LIN {X 87.779,Y 86.082,Z 65.500,A 180.000,B 0.000,C 180.000} C_DIS
LIN {X 87.601,Y 86.233,Z 65.500,A 180.000,B 0.000,C 180.000} C_DIS
LIN {X 87.468,Y 86.349,Z 65.500,A 180.000,B 0.000,C 180.000} C_DIS
LIN {X 87.422,Y 86.393,Z 65.500,A 180.000,B 0.000,C 180.000} C_DIS
LIN {X 87.064,Y 86.731,Z 65.500,A 180.000,B 0.000,C 180.000} C_DIS
LIN {X 86.901,Y 86.885,Z 65.500,A 180.000,B 0.000,C 180.000} C_DIS
LIN {X 86.885,Y 86.901,Z 65.500,A 180.000,B 0.000,C 180.000} C_DIS
LIN {X 86.731,Y 87.064,Z 65.500,A 180.000,B 0.000,C 180.000} C_DIS
LIN {X 86.393,Y 87.422,Z 65.500,A 180.000,B 0.000,C 180.000} C_DIS
LIN {X 86.349,Y 87.468,Z 65.500,A 180.000,B 0.000,C 180.000} C_DIS
LIN {X 86.233,Y 87.601,Z 65.500,A 180.000,B 0.000,C 180.000} C_DIS
LIN {X 85.931,Y 87.958,Z 65.500,A 180.000,B 0.000,C 180.000} C_DIS
LIN {X 85.813,Y 88.098,Z 65.500,A 180.000,B 0.000,C 180.000} C_DIS
LIN {X 85.781,Y 88.137,Z 65.500,A 180.000,B 0.000,C 180.000} C_DIS
LIN {X 85.645,Y 88.316,Z 65.500,A 180.000,B 0.000,C 180.000} C_DIS
LIN {X 85.376,Y 88.673,Z 65.500,A 180.000,B 0.000,C 180.000} C_DIS
LIN {X 85.276,Y 88.806,Z 65.500,A 180.000,B 0.000,C 180.000} C_DIS
LIN {X 85.244,Y 88.852,Z 65.500,A 180.000,B 0.000,C 180.000} C_DIS
LIN {X 85.125,Y 89.031,Z 65.500,A 180.000,B 0.000,C 180.000} C_DIS
LIN {X 84.886,Y 89.388,Z 65.500,A 180.000,B 0.000,C 180.000} C_DIS
LIN {X 84.770,Y 89.567,Z 65.500,A 180.000,B 0.000,C 180.000} C_DIS
LIN {X 84.740,Y 89.618,Z 65.500,A 180.000,B 0.000,C 180.000} C_DIS
LIN {X 84.454,Y 90.103,Z 65.500,A 180.000,B 0.000,C 180.000} C_DIS
LIN {X 84.383,Y 90.225,Z 65.500,A 180.000,B 0.000,C 180.000} C_DIS
LIN {X 84.351,Y 90.282,Z 65.500,A 180.000,B 0.000,C 180.000} C_DIS
LIN {X 84.259,Y 90.461,Z 65.500,A 180.000,B 0.000,C 180.000} C_DIS
LIN {X 84.025,Y 90.913,Z 65.500,A 180.000,B 0.000,C 180.000} C_DIS
LIN {X 83.983,Y 90.997,Z 65.500,A 180.000,B 0.000,C 180.000} C_DIS
LIN {X 83.902,Y 91.176,Z 65.500,A 180.000,B 0.000,C 180.000} C_DIS
LIN {X 83.668,Y 91.700,Z 65.500,A 180.000,B 0.000,C 180.000} C_DIS
LIN {X 83.662,Y 91.712,Z 65.500,A 180.000,B 0.000,C 180.000} C_DIS
LIN {X 83.591,Y 91.891,Z 65.500,A 180.000,B 0.000,C 180.000} C_DIS
LIN {X 83.386,Y 92.427,Z 65.500,A 180.000,B 0.000,C 180.000} C_DIS
LIN {X 83.322,Y 92.606,Z 65.500,A 180.000,B 0.000,C 180.000} C_DIS
LIN {X 83.310,Y 92.642,Z 65.500,A 180.000,B 0.000,C 180.000} C_DIS
LIN {X 83.131,Y 93.203,Z 65.500,A 180.000,B 0.000,C 180.000} C_DIS
LIN {X 83.094,Y 93.321,Z 65.500,A 180.000,B 0.000,C 180.000} C_DIS
LIN {X 83.046,Y 93.500,Z 65.500,A 180.000,B 0.000,C 180.000} C_DIS
LIN {X 82.908,Y 94.036,Z 65.500,A 180.000,B 0.000,C 180.000} C_DIS
LIN {X 82.865,Y 94.215,Z 65.500,A 180.000,B 0.000,C 180.000} C_DIS
LIN {X 82.829,Y 94.394,Z 65.500,A 180.000,B 0.000,C 180.000} C_DIS
LIN {X 82.758,Y 94.751,Z 65.500,A 180.000,B 0.000,C 180.000} C_DIS
LIN {X 82.722,Y 94.930,Z 65.500,A 180.000,B 0.000,C 180.000} C_DIS
LIN {X 82.694,Y 95.109,Z 65.500,A 180.000,B 0.000,C 180.000} C_DIS
LIN {X 82.618,Y 95.645,Z 65.500,A 180.000,B 0.000,C 180.000} C_DIS
LIN {X 82.595,Y 95.815,Z 65.500,A 180.000,B 0.000,C 180.000} C_DIS
LIN {X 82.594,Y 95.824,Z 65.500,A 180.000,B 0.000,C 180.000} C_DIS
LIN {X 82.578,Y 96.003,Z 65.500,A 180.000,B 0.000,C 180.000} C_DIS
LIN {X 82.533,Y 96.539,Z 65.500,A 180.000,B 0.000,C 180.000} C_DIS
LIN {X 82.521,Y 96.718,Z 65.500,A 180.000,B 0.000,C 180.000} C_DIS
LIN {X 82.516,Y 96.897,Z 65.500,A 180.000,B 0.000,C 180.000} C_DIS
LIN {X 82.501,Y 97.433,Z 65.500,A 180.000,B 0.000,C 180.000} C_DIS
LIN {X 82.502,Y 97.612,Z 65.500,A 180.000,B 0.000,C 180.000} C_DIS
LIN {X 82.517,Y 98.148,Z 65.500,A 180.000,B 0.000,C 180.000} C_DIS
LIN {X 82.523,Y 98.327,Z 65.500,A 180.000,B 0.000,C 180.000} C_DIS
LIN {X 82.536,Y 98.505,Z 65.500,A 180.000,B 0.000,C 180.000} C_DIS
LIN {X 82.582,Y 99.042,Z 65.500,A 180.000,B 0.000,C 180.000} C_DIS
LIN {X 82.595,Y 99.185,Z 65.500,A 180.000,B 0.000,C 180.000} C_DIS
LIN {X 82.599,Y 99.221,Z 65.500,A 180.000,B 0.000,C 180.000} C_DIS
LIN {X 82.624,Y 99.399,Z 65.500,A 180.000,B 0.000,C 180.000} C_DIS
LIN {X 82.700,Y 99.936,Z 65.500,A 180.000,B 0.000,C 180.000} C_DIS
LIN {X 82.731,Y 100.114,Z 65.500,A 180.000,B 0.000,C 180.000} C_DIS
LIN {X 82.838,Y 100.651,Z 65.500,A 180.000,B 0.000,C 180.000} C_DIS
LIN {X 82.874,Y 100.829,Z 65.500,A 180.000,B 0.000,C 180.000} C_DIS
LIN {X 82.919,Y 101.008,Z 65.500,A 180.000,B 0.000,C 180.000} C_DIS
LIN {X 83.057,Y 101.545,Z 65.500,A 180.000,B 0.000,C 180.000} C_DIS
LIN {X 83.108,Y 101.723,Z 65.500,A 180.000,B 0.000,C 180.000} C_DIS
LIN {X 83.310,Y 102.358,Z 65.500,A 180.000,B 0.000,C 180.000} C_DIS
LIN {X 83.336,Y 102.438,Z 65.500,A 180.000,B 0.000,C 180.000} C_DIS
LIN {X 83.403,Y 102.617,Z 65.500,A 180.000,B 0.000,C 180.000} C_DIS
LIN {X 83.608,Y 103.153,Z 65.500,A 180.000,B 0.000,C 180.000} C_DIS
LIN {X 83.668,Y 103.300,Z 65.500,A 180.000,B 0.000,C 180.000} C_DIS
LIN {X 83.922,Y 103.869,Z 65.500,A 180.000,B 0.000,C 180.000} C_DIS
LIN {X 84.005,Y 104.047,Z 65.500,A 180.000,B 0.000,C 180.000} C_DIS
LIN {X 84.025,Y 104.087,Z 65.500,A 180.000,B 0.000,C 180.000} C_DIS
LIN {X 84.282,Y 104.584,Z 65.500,A 180.000,B 0.000,C 180.000} C_DIS
LIN {X 84.375,Y 104.762,Z 65.500,A 180.000,B 0.000,C 180.000} C_DIS
LIN {X 84.383,Y 104.775,Z 65.500,A 180.000,B 0.000,C 180.000} C_DIS
LIN {X 84.480,Y 104.941,Z 65.500,A 180.000,B 0.000,C 180.000} C_DIS
LIN {X 84.740,Y 105.382,Z 65.500,A 180.000,B 0.000,C 180.000} C_DIS
LIN {X 84.797,Y 105.477,Z 65.500,A 180.000,B 0.000,C 180.000} C_DIS
LIN {X 84.915,Y 105.656,Z 65.500,A 180.000,B 0.000,C 180.000} C_DIS
LIN {X 85.154,Y 106.014,Z 65.500,A 180.000,B 0.000,C 180.000} C_DIS
LIN {X 85.276,Y 106.193,Z 65.500,A 180.000,B 0.000,C 180.000} C_DIS
LIN {X 85.276,Y 106.194,Z 65.500,A 180.000,B 0.000,C 180.000} C_DIS
LIN {X 85.409,Y 106.371,Z 65.500,A 180.000,B 0.000,C 180.000} C_DIS
LIN {X 85.678,Y 106.729,Z 65.500,A 180.000,B 0.000,C 180.000} C_DIS
LIN {X 85.813,Y 106.902,Z 65.500,A 180.000,B 0.000,C 180.000} C_DIS
LIN {X 85.818,Y 106.908,Z 65.500,A 180.000,B 0.000,C 180.000} C_DIS
LIN {X 86.271,Y 107.444,Z 65.500,A 180.000,B 0.000,C 180.000} C_DIS
LIN {X 86.349,Y 107.532,Z 65.500,A 180.000,B 0.000,C 180.000} C_DIS
LIN {X 86.435,Y 107.623,Z 65.500,A 180.000,B 0.000,C 180.000} C_DIS
LIN {X 86.773,Y 107.980,Z 65.500,A 180.000,B 0.000,C 180.000} C_DIS
LIN {X 86.885,Y 108.099,Z 65.500,A 180.000,B 0.000,C 180.000} C_DIS
LIN {X 86.947,Y 108.159,Z 65.500,A 180.000,B 0.000,C 180.000} C_DIS
LIN {X 87.422,Y 108.607,Z 65.500,A 180.000,B 0.000,C 180.000} C_DIS
LIN {X 87.517,Y 108.695,Z 65.500,A 180.000,B 0.000,C 180.000} C_DIS
LIN {X 87.601,Y 108.767,Z 65.500,A 180.000,B 0.000,C 180.000} C_DIS
LIN {X 87.958,Y 109.069,Z 65.500,A 180.000,B 0.000,C 180.000} C_DIS
LIN {X 88.137,Y 109.219,Z 65.500,A 180.000,B 0.000,C 180.000} C_DIS
LIN {X 88.153,Y 109.232,Z 65.500,A 180.000,B 0.000,C 180.000} C_DIS
LIN {X 88.316,Y 109.355,Z 65.500,A 180.000,B 0.000,C 180.000} C_DIS
LIN {X 88.673,Y 109.624,Z 65.500,A 180.000,B 0.000,C 180.000} C_DIS
LIN {X 88.852,Y 109.756,Z 65.500,A 180.000,B 0.000,C 180.000} C_DIS
LIN {X 88.870,Y 109.768,Z 65.500,A 180.000,B 0.000,C 180.000} C_DIS
LIN {X 89.031,Y 109.875,Z 65.500,A 180.000,B 0.000,C 180.000} C_DIS
LIN {X 89.405,Y 110.126,Z 65.500,A 180.000,B 0.000,C 180.000} C_DIS
LIN {X 89.567,Y 110.230,Z 65.500,A 180.000,B 0.000,C 180.000} C_DIS
LIN {X 89.693,Y 110.304,Z 65.500,A 180.000,B 0.000,C 180.000} C_DIS
LIN {X 90.103,Y 110.546,Z 65.500,A 180.000,B 0.000,C 180.000} C_DIS
LIN {X 90.282,Y 110.649,Z 65.500,A 180.000,B 0.000,C 180.000} C_DIS
LIN {X 90.307,Y 110.662,Z 65.500,A 180.000,B 0.000,C 180.000} C_DIS
LIN {X 90.818,Y 110.926,Z 65.500,A 180.000,B 0.000,C 180.000} C_DIS
LIN {X 90.997,Y 111.017,Z 65.500,A 180.000,B 0.000,C 180.000} C_DIS
LIN {X 91.002,Y 111.019,Z 65.500,A 180.000,B 0.000,C 180.000} C_DIS
LIN {X 91.176,Y 111.098,Z 65.500,A 180.000,B 0.000,C 180.000} C_DIS
LIN {X 91.533,Y 111.258,Z 65.500,A 180.000,B 0.000,C 180.000} C_DIS
LIN {X 91.712,Y 111.338,Z 65.500,A 180.000,B 0.000,C 180.000} C_DIS
LIN {X 91.806,Y 111.377,Z 65.500,A 180.000,B 0.000,C 180.000} C_DIS
LIN {X 91.891,Y 111.409,Z 65.500,A 180.000,B 0.000,C 180.000} C_DIS
LIN {X 92.427,Y 111.614,Z 65.500,A 180.000,B 0.000,C 180.000} C_DIS
LIN {X 92.606,Y 111.678,Z 65.500,A 180.000,B 0.000,C 180.000} C_DIS
LIN {X 92.964,Y 111.792,Z 65.500,A 180.000,B 0.000,C 180.000} C_DIS
LIN {X 93.142,Y 111.849,Z 65.500,A 180.000,B 0.000,C 180.000} C_DIS
LIN {X 93.321,Y 111.906,Z 65.500,A 180.000,B 0.000,C 180.000} C_DIS
LIN {X 93.346,Y 111.913,Z 65.500,A 180.000,B 0.000,C 180.000} C_DIS
LIN {X 93.500,Y 111.954,Z 65.500,A 180.000,B 0.000,C 180.000} C_DIS
LIN {X 94.036,Y 112.092,Z 65.500,A 180.000,B 0.000,C 180.000} C_DIS
LIN {X 94.215,Y 112.135,Z 65.500,A 180.000,B 0.000,C 180.000} C_DIS
LIN {X 94.394,Y 112.171,Z 65.500,A 180.000,B 0.000,C 180.000} C_DIS
LIN {X 94.895,Y 112.271,Z 65.500,A 180.000,B 0.000,C 180.000} C_DIS
LIN {X 94.930,Y 112.278,Z 65.500,A 180.000,B 0.000,C 180.000} C_DIS
LIN {X 95.109,Y 112.306,Z 65.500,A 180.000,B 0.000,C 180.000} C_DIS
LIN {X 95.645,Y 112.382,Z 65.500,A 180.000,B 0.000,C 180.000} C_DIS
LIN {X 95.824,Y 112.406,Z 65.500,A 180.000,B 0.000,C 180.000} C_DIS
LIN {X 96.003,Y 112.422,Z 65.500,A 180.000,B 0.000,C 180.000} C_DIS
LIN {X 96.539,Y 112.467,Z 65.500,A 180.000,B 0.000,C 180.000} C_DIS
LIN {X 96.718,Y 112.479,Z 65.500,A 180.000,B 0.000,C 180.000} C_DIS
LIN {X 96.897,Y 112.484,Z 65.500,A 180.000,B 0.000,C 180.000} C_DIS
LIN {X 97.433,Y 112.499,Z 65.500,A 180.000,B 0.000,C 180.000} C_DIS
LIN {X 97.612,Y 112.498,Z 65.500,A 180.000,B 0.000,C 180.000} C_DIS
LIN {X 98.148,Y 112.483,Z 65.500,A 180.000,B 0.000,C 180.000} C_DIS
LIN {X 98.327,Y 112.477,Z 65.500,A 180.000,B 0.000,C 180.000} C_DIS
LIN {X 98.505,Y 112.464,Z 65.500,A 180.000,B 0.000,C 180.000} C_DIS
LIN {X 99.042,Y 112.418,Z 65.500,A 180.000,B 0.000,C 180.000} C_DIS
LIN {X 99.221,Y 112.401,Z 65.500,A 180.000,B 0.000,C 180.000} C_DIS
LIN {X 99.399,Y 112.376,Z 65.500,A 180.000,B 0.000,C 180.000} C_DIS
LIN {X 99.936,Y 112.300,Z 65.500,A 180.000,B 0.000,C 180.000} C_DIS
LIN {X 100.105,Y 112.271,Z 65.500,A 180.000,B 0.000,C 180.000} C_DIS
LIN {X 100.651,Y 112.162,Z 65.500,A 180.000,B 0.000,C 180.000} C_DIS
LIN {X 100.829,Y 112.126,Z 65.500,A 180.000,B 0.000,C 180.000} C_DIS
LIN {X 100.966,Y 112.092,Z 65.500,A 180.000,B 0.000,C 180.000} C_DIS
LIN {X 101.545,Y 111.943,Z 65.500,A 180.000,B 0.000,C 180.000} C_DIS
LIN {X 101.654,Y 111.913,Z 65.500,A 180.000,B 0.000,C 180.000} C_DIS
LIN {X 101.723,Y 111.892,Z 65.500,A 180.000,B 0.000,C 180.000} C_DIS
LIN {X 102.260,Y 111.721,Z 65.500,A 180.000,B 0.000,C 180.000} C_DIS
LIN {X 102.438,Y 111.664,Z 65.500,A 180.000,B 0.000,C 180.000} C_DIS
LIN {X 102.617,Y 111.597,Z 65.500,A 180.000,B 0.000,C 180.000} C_DIS
LIN {X 103.153,Y 111.392,Z 65.500,A 180.000,B 0.000,C 180.000} C_DIS
LIN {X 103.194,Y 111.377,Z 65.500,A 180.000,B 0.000,C 180.000} C_DIS
LIN {X 103.332,Y 111.318,Z 65.500,A 180.000,B 0.000,C 180.000} C_DIS
LIN {X 103.869,Y 111.078,Z 65.500,A 180.000,B 0.000,C 180.000} C_DIS
LIN {X 103.998,Y 111.019,Z 65.500,A 180.000,B 0.000,C 180.000} C_DIS
LIN {X 104.047,Y 110.995,Z 65.500,A 180.000,B 0.000,C 180.000} C_DIS
LIN {X 104.226,Y 110.903,Z 65.500,A 180.000,B 0.000,C 180.000} C_DIS
LIN {X 104.693,Y 110.662,Z 65.500,A 180.000,B 0.000,C 180.000} C_DIS
LIN {X 104.762,Y 110.625,Z 65.500,A 180.000,B 0.000,C 180.000} C_DIS
LIN {X 104.941,Y 110.520,Z 65.500,A 180.000,B 0.000,C 180.000} C_DIS
LIN {X 105.307,Y 110.304,Z 65.500,A 180.000,B 0.000,C 180.000} C_DIS
LIN {X 105.477,Y 110.203,Z 65.500,A 180.000,B 0.000,C 180.000} C_DIS
LIN {X 105.595,Y 110.126,Z 65.500,A 180.000,B 0.000,C 180.000} C_DIS
LIN {X 106.014,Y 109.846,Z 65.500,A 180.000,B 0.000,C 180.000} C_DIS
LIN {X 106.130,Y 109.768,Z 65.500,A 180.000,B 0.000,C 180.000} C_DIS
LIN {X 106.193,Y 109.724,Z 65.500,A 180.000,B 0.000,C 180.000} C_DIS
LIN {X 106.371,Y 109.591,Z 65.500,A 180.000,B 0.000,C 180.000} C_DIS
LIN {X 106.729,Y 109.322,Z 65.500,A 180.000,B 0.000,C 180.000} C_DIS
LIN {X 106.847,Y 109.232,Z 65.500,A 180.000,B 0.000,C 180.000} C_DIS
LIN {X 106.908,Y 109.182,Z 65.500,A 180.000,B 0.000,C 180.000} C_DIS
LIN {X 107.444,Y 108.729,Z 65.500,A 180.000,B 0.000,C 180.000} C_DIS
LIN {X 107.483,Y 108.695,Z 65.500,A 180.000,B 0.000,C 180.000} C_DIS
LIN {X 107.623,Y 108.565,Z 65.500,A 180.000,B 0.000,C 180.000} C_DIS
LIN {X 108.053,Y 108.159,Z 65.500,A 180.000,B 0.000,C 180.000} C_DIS
LIN {X 108.159,Y 108.053,Z 65.500,A 180.000,B 0.000,C 180.000} C_DIS
LIN {X 108.565,Y 107.623,Z 65.500,A 180.000,B 0.000,C 180.000} C_DIS
LIN {X 108.695,Y 107.483,Z 65.500,A 180.000,B 0.000,C 180.000} C_DIS
LIN {X 108.729,Y 107.444,Z 65.500,A 180.000,B 0.000,C 180.000} C_DIS
LIN {X 109.182,Y 106.908,Z 65.500,A 180.000,B 0.000,C 180.000} C_DIS
LIN {X 109.232,Y 106.847,Z 65.500,A 180.000,B 0.000,C 180.000} C_DIS
LIN {X 109.322,Y 106.729,Z 65.500,A 180.000,B 0.000,C 180.000} C_DIS
LIN {X 109.591,Y 106.371,Z 65.500,A 180.000,B 0.000,C 180.000} C_DIS
LIN {X 109.724,Y 106.193,Z 65.500,A 180.000,B 0.000,C 180.000} C_DIS
LIN {X 109.768,Y 106.130,Z 65.500,A 180.000,B 0.000,C 180.000} C_DIS
LIN {X 109.846,Y 106.014,Z 65.500,A 180.000,B 0.000,C 180.000} C_DIS
LIN {X 110.126,Y 105.595,Z 65.500,A 180.000,B 0.000,C 180.000} C_DIS
LIN {X 110.203,Y 105.477,Z 65.500,A 180.000,B 0.000,C 180.000} C_DIS
LIN {X 110.304,Y 105.307,Z 65.500,A 180.000,B 0.000,C 180.000} C_DIS
LIN {X 110.520,Y 104.941,Z 65.500,A 180.000,B 0.000,C 180.000} C_DIS
LIN {X 110.625,Y 104.762,Z 65.500,A 180.000,B 0.000,C 180.000} C_DIS
LIN {X 110.662,Y 104.693,Z 65.500,A 180.000,B 0.000,C 180.000} C_DIS
LIN {X 110.903,Y 104.226,Z 65.500,A 180.000,B 0.000,C 180.000} C_DIS
LIN {X 110.995,Y 104.047,Z 65.500,A 180.000,B 0.000,C 180.000} C_DIS
LIN {X 111.019,Y 103.998,Z 65.500,A 180.000,B 0.000,C 180.000} C_DIS
LIN {X 111.078,Y 103.869,Z 65.500,A 180.000,B 0.000,C 180.000} C_DIS
LIN {X 111.318,Y 103.332,Z 65.500,A 180.000,B 0.000,C 180.000} C_DIS
LIN {X 111.377,Y 103.194,Z 65.500,A 180.000,B 0.000,C 180.000} C_DIS
LIN {X 111.392,Y 103.153,Z 65.500,A 180.000,B 0.000,C 180.000} C_DIS
LIN {X 111.597,Y 102.617,Z 65.500,A 180.000,B 0.000,C 180.000} C_DIS
LIN {X 111.664,Y 102.438,Z 65.500,A 180.000,B 0.000,C 180.000} C_DIS
LIN {X 111.721,Y 102.260,Z 65.500,A 180.000,B 0.000,C 180.000} C_DIS
LIN {X 111.892,Y 101.723,Z 65.500,A 180.000,B 0.000,C 180.000} C_DIS
LIN {X 111.913,Y 101.654,Z 65.500,A 180.000,B 0.000,C 180.000} C_DIS
LIN {X 111.943,Y 101.545,Z 65.500,A 180.000,B 0.000,C 180.000} C_DIS
LIN {X 112.092,Y 100.966,Z 65.500,A 180.000,B 0.000,C 180.000} C_DIS
LIN {X 112.126,Y 100.829,Z 65.500,A 180.000,B 0.000,C 180.000} C_DIS
LIN {X 112.162,Y 100.651,Z 65.500,A 180.000,B 0.000,C 180.000} C_DIS
LIN {X 112.271,Y 100.105,Z 65.500,A 180.000,B 0.000,C 180.000} C_DIS
LIN {X 112.300,Y 99.936,Z 65.500,A 180.000,B 0.000,C 180.000} C_DIS
LIN {X 112.376,Y 99.399,Z 65.500,A 180.000,B 0.000,C 180.000} C_DIS
LIN {X 112.401,Y 99.221,Z 65.500,A 180.000,B 0.000,C 180.000} C_DIS
LIN {X 112.418,Y 99.042,Z 65.500,A 180.000,B 0.000,C 180.000} C_DIS
LIN {X 112.464,Y 98.505,Z 65.500,A 180.000,B 0.000,C 180.000} C_DIS
LIN {X 112.477,Y 98.327,Z 65.500,A 180.000,B 0.000,C 180.000} C_DIS
LIN {X 112.483,Y 98.148,Z 65.500,A 180.000,B 0.000,C 180.000} C_DIS
LIN {X 112.498,Y 97.612,Z 65.500,A 180.000,B 0.000,C 180.000} C_DIS
LIN {X 112.499,Y 97.433,Z 65.500,A 180.000,B 0.000,C 180.000} C_DIS
LIN {X 112.484,Y 96.897,Z 65.500,A 180.000,B 0.000,C 180.000} C_DIS
LIN {X 112.479,Y 96.718,Z 65.500,A 180.000,B 0.000,C 180.000} C_DIS
LIN {X 112.467,Y 96.539,Z 65.500,A 180.000,B 0.000,C 180.000} C_DIS
LIN {X 112.422,Y 96.003,Z 65.500,A 180.000,B 0.000,C 180.000} C_DIS
LIN {X 112.406,Y 95.824,Z 65.500,A 180.000,B 0.000,C 180.000} C_DIS
LIN {X 112.382,Y 95.645,Z 65.500,A 180.000,B 0.000,C 180.000} C_DIS
LIN {X 112.306,Y 95.109,Z 65.500,A 180.000,B 0.000,C 180.000} C_DIS
LIN {X 112.278,Y 94.930,Z 65.500,A 180.000,B 0.000,C 180.000} C_DIS
LIN {X 112.271,Y 94.895,Z 65.500,A 180.000,B 0.000,C 180.000} C_DIS
LIN {X 112.171,Y 94.394,Z 65.500,A 180.000,B 0.000,C 180.000} C_DIS
LIN {X 112.135,Y 94.215,Z 65.500,A 180.000,B 0.000,C 180.000} C_DIS
LIN {X 112.092,Y 94.036,Z 65.500,A 180.000,B 0.000,C 180.000} C_DIS
LIN {X 111.954,Y 93.500,Z 65.500,A 180.000,B 0.000,C 180.000} C_DIS
LIN {X 111.913,Y 93.346,Z 65.500,A 180.000,B 0.000,C 180.000} C_DIS
LIN {X 111.906,Y 93.321,Z 65.500,A 180.000,B 0.000,C 180.000} C_DIS
LIN {X 111.849,Y 93.142,Z 65.500,A 180.000,B 0.000,C 180.000} C_DIS
LIN {X 111.734,Y 92.782,Z 65.500,A 180.000,B 0.000,C 180.000} C_DIS
LIN {X 111.678,Y 92.606,Z 65.500,A 180.000,B 0.000,C 180.000} C_DIS
LIN {X 111.614,Y 92.427,Z 65.500,A 180.000,B 0.000,C 180.000} C_DIS
LIN {X 111.409,Y 91.891,Z 65.500,A 180.000,B 0.000,C 180.000} C_DIS
LIN {X 111.377,Y 91.806,Z 65.500,A 180.000,B 0.000,C 180.000} C_DIS
LIN {X 111.338,Y 91.712,Z 65.500,A 180.000,B 0.000,C 180.000} C_DIS
LIN {X 111.258,Y 91.533,Z 65.500,A 180.000,B 0.000,C 180.000} C_DIS
LIN {X 111.098,Y 91.176,Z 65.500,A 180.000,B 0.000,C 180.000} C_DIS
LIN {X 111.019,Y 91.002,Z 65.500,A 180.000,B 0.000,C 180.000} C_DIS
LIN {X 111.017,Y 90.997,Z 65.500,A 180.000,B 0.000,C 180.000} C_DIS
LIN {X 110.946,Y 90.857,Z 65.500,A 180.000,B 0.000,C 180.000} C_DIS
; Link Move Starts
LIN {X 110.802,Y 90.577,Z 65.500,A 180.000,B 0.000,C 180.000} C_DIS
LIN {X 110.657,Y 90.297,Z 65.499,A 180.000,B 0.000,C 180.000} C_DIS
LIN {X 110.500,Y 90.024,Z 65.498,A 180.000,B 0.000,C 180.000} C_DIS
LIN {X 110.340,Y 89.753,Z 65.496,A 180.000,B 0.000,C 180.000} C_DIS
LIN {X 110.178,Y 89.483,Z 65.494,A 180.000,B 0.000,C 180.000} C_DIS
LIN {X 110.003,Y 89.221,Z 65.491,A 180.000,B 0.000,C 180.000} C_DIS
LIN {X 109.828,Y 88.959,Z 65.488,A 180.000,B 0.000,C 180.000} C_DIS
LIN {X 109.646,Y 88.702,Z 65.485,A 180.000,B 0.000,C 180.000} C_DIS
LIN {X 109.457,Y 88.450,Z 65.481,A 180.000,B 0.000,C 180.000} C_DIS
LIN {X 109.267,Y 88.199,Z 65.477,A 180.000,B 0.000,C 180.000} C_DIS
LIN {X 109.067,Y 87.956,Z 65.472,A 180.000,B 0.000,C 180.000} C_DIS
LIN {X 108.965,Y 87.835,Z 65.469,A 180.000,B 0.000,C 180.000} C_DIS
LIN {X 108.863,Y 87.715,Z 65.467,A 180.000,B 0.000,C 180.000} C_DIS
LIN {X 108.762,Y 87.595,Z 65.464,A 180.000,B 0.000,C 180.000} C_DIS
LIN {X 108.658,Y 87.476,Z 65.461,A 180.000,B 0.000,C 180.000} C_DIS
LIN {X 108.550,Y 87.361,Z 65.459,A 180.000,B 0.000,C 180.000} C_DIS
LIN {X 108.442,Y 87.247,Z 65.456,A 180.000,B 0.000,C 180.000} C_DIS
LIN {X 108.334,Y 87.132,Z 65.452,A 180.000,B 0.000,C 180.000} C_DIS
LIN {X 108.226,Y 87.018,Z 65.449,A 180.000,B 0.000,C 180.000} C_DIS
LIN {X 108.117,Y 86.904,Z 65.446,A 180.000,B 0.000,C 180.000} C_DIS
LIN {X 108.004,Y 86.795,Z 65.443,A 180.000,B 0.000,C 180.000} C_DIS
LIN {X 107.889,Y 86.687,Z 65.439,A 180.000,B 0.000,C 180.000} C_DIS
LIN {X 107.775,Y 86.578,Z 65.436,A 180.000,B 0.000,C 180.000} C_DIS
LIN {X 107.660,Y 86.470,Z 65.432,A 180.000,B 0.000,C 180.000} C_DIS
LIN {X 107.546,Y 86.362,Z 65.428,A 180.000,B 0.000,C 180.000} C_DIS
LIN {X 107.428,Y 86.257,Z 65.425,A 180.000,B 0.000,C 180.000} C_DIS
LIN {X 107.308,Y 86.156,Z 65.421,A 180.000,B 0.000,C 180.000} C_DIS
LIN {X 107.187,Y 86.054,Z 65.417,A 180.000,B 0.000,C 180.000} C_DIS
LIN {X 107.067,Y 85.953,Z 65.413,A 180.000,B 0.000,C 180.000} C_DIS
LIN {X 106.947,Y 85.851,Z 65.409,A 180.000,B 0.000,C 180.000} C_DIS
LIN {X 106.825,Y 85.751,Z 65.405,A 180.000,B 0.000,C 180.000} C_DIS
LIN {X 106.699,Y 85.656,Z 65.400,A 180.000,B 0.000,C 180.000} C_DIS
LIN {X 106.573,Y 85.561,Z 65.396,A 180.000,B 0.000,C 180.000} C_DIS
LIN {X 106.448,Y 85.467,Z 65.392,A 180.000,B 0.000,C 180.000} C_DIS
LIN {X 106.322,Y 85.372,Z 65.387,A 180.000,B 0.000,C 180.000} C_DIS
LIN {X 106.196,Y 85.278,Z 65.383,A 180.000,B 0.000,C 180.000} C_DIS
LIN {X 106.066,Y 85.189,Z 65.378,A 180.000,B 0.000,C 180.000} C_DIS
LIN {X 105.935,Y 85.101,Z 65.373,A 180.000,B 0.000,C 180.000} C_DIS
LIN {X 105.804,Y 85.014,Z 65.369,A 180.000,B 0.000,C 180.000} C_DIS
LIN {X 105.673,Y 84.926,Z 65.364,A 180.000,B 0.000,C 180.000} C_DIS
LIN {X 105.542,Y 84.839,Z 65.359,A 180.000,B 0.000,C 180.000} C_DIS
LIN {X 105.408,Y 84.755,Z 65.354,A 180.000,B 0.000,C 180.000} C_DIS
LIN {X 105.340,Y 84.715,Z 65.351,A 180.000,B 0.000,C 180.000} C_DIS
LIN {X 105.273,Y 84.675,Z 65.349,A 180.000,B 0.000,C 180.000} C_DIS
LIN {X 105.205,Y 84.635,Z 65.346,A 180.000,B 0.000,C 180.000} C_DIS
LIN {X 105.137,Y 84.595,Z 65.344,A 180.000,B 0.000,C 180.000} C_DIS
LIN {X 105.069,Y 84.555,Z 65.341,A 180.000,B 0.000,C 180.000} C_DIS
LIN {X 105.001,Y 84.515,Z 65.339,A 180.000,B 0.000,C 180.000} C_DIS
LIN {X 104.933,Y 84.475,Z 65.336,A 180.000,B 0.000,C 180.000} C_DIS
LIN {X 104.866,Y 84.435,Z 65.333,A 180.000,B 0.000,C 180.000} C_DIS
LIN {X 104.798,Y 84.395,Z 65.331,A 180.000,B 0.000,C 180.000} C_DIS
LIN {X 104.729,Y 84.357,Z 65.328,A 180.000,B 0.000,C 180.000} C_DIS
LIN {X 104.659,Y 84.321,Z 65.325,A 180.000,B 0.000,C 180.000} C_DIS
LIN {X 104.519,Y 84.248,Z 65.320,A 180.000,B 0.000,C 180.000} C_DIS
LIN {X 104.379,Y 84.176,Z 65.315,A 180.000,B 0.000,C 180.000} C_DIS
LIN {X 104.239,Y 84.104,Z 65.309,A 180.000,B 0.000,C 180.000} C_DIS
LIN {X 104.169,Y 84.068,Z 65.307,A 180.000,B 0.000,C 180.000} C_DIS
LIN {X 104.099,Y 84.031,Z 65.304,A 180.000,B 0.000,C 180.000} C_DIS
LIN {X 104.029,Y 83.996,Z 65.301,A 180.000,B 0.000,C 180.000} C_DIS
LIN {X 103.958,Y 83.962,Z 65.298,A 180.000,B 0.000,C 180.000} C_DIS
LIN {X 103.886,Y 83.930,Z 65.296,A 180.000,B 0.000,C 180.000} C_DIS
LIN {X 103.742,Y 83.865,Z 65.290,A 180.000,B 0.000,C 180.000} C_DIS
LIN {X 103.527,Y 83.769,Z 65.282,A 180.000,B 0.000,C 180.000} C_DIS
LIN {X 103.383,Y 83.705,Z 65.276,A 180.000,B 0.000,C 180.000} C_DIS
LIN {X 103.311,Y 83.672,Z 65.274,A 180.000,B 0.000,C 180.000} C_DIS
LIN {X 103.239,Y 83.641,Z 65.271,A 180.000,B 0.000,C 180.000} C_DIS
LIN {X 103.166,Y 83.612,Z 65.268,A 180.000,B 0.000,C 180.000} C_DIS
LIN {X 102.945,Y 83.528,Z 65.260,A 180.000,B 0.000,C 180.000} C_DIS
LIN {X 102.798,Y 83.472,Z 65.254,A 180.000,B 0.000,C 180.000} C_DIS
LIN {X 102.724,Y 83.444,Z 65.252,A 180.000,B 0.000,C 180.000} C_DIS
LIN {X 102.577,Y 83.388,Z 65.246,A 180.000,B 0.000,C 180.000} C_DIS
LIN {X 102.503,Y 83.360,Z 65.243,A 180.000,B 0.000,C 180.000} C_DIS
LIN {X 102.429,Y 83.333,Z 65.241,A 180.000,B 0.000,C 180.000} C_DIS
LIN {X 102.354,Y 83.309,Z 65.238,A 180.000,B 0.000,C 180.000} C_DIS
LIN {X 102.204,Y 83.261,Z 65.232,A 180.000,B 0.000,C 180.000} C_DIS
LIN {X 102.129,Y 83.237,Z 65.230,A 180.000,B 0.000,C 180.000} C_DIS
LIN {X 101.979,Y 83.189,Z 65.224,A 180.000,B 0.000,C 180.000} C_DIS
LIN {X 101.754,Y 83.118,Z 65.216,A 180.000,B 0.000,C 180.000} C_DIS
LIN {X 101.679,Y 83.094,Z 65.213,A 180.000,B 0.000,C 180.000} C_DIS
LIN {X 101.603,Y 83.073,Z 65.210,A 180.000,B 0.000,C 180.000} C_DIS
LIN {X 101.527,Y 83.053,Z 65.208,A 180.000,B 0.000,C 180.000} C_DIS
LIN {X 101.374,Y 83.013,Z 65.202,A 180.000,B 0.000,C 180.000} C_DIS
LIN {X 100.917,Y 82.895,Z 65.186,A 180.000,B 0.000,C 180.000} C_DIS
LIN {X 100.840,Y 82.877,Z 65.183,A 180.000,B 0.000,C 180.000} C_DIS
LIN {X 100.763,Y 82.860,Z 65.180,A 180.000,B 0.000,C 180.000} C_DIS
LIN {X 100.223,Y 82.753,Z 65.161,A 180.000,B 0.000,C 180.000} C_DIS
LIN {X 100.145,Y 82.737,Z 65.158,A 180.000,B 0.000,C 180.000} C_DIS
LIN {X 100.068,Y 82.722,Z 65.155,A 180.000,B 0.000,C 180.000} C_DIS
LIN {X 99.991,Y 82.708,Z 65.153,A 180.000,B 0.000,C 180.000} C_DIS
LIN {X 99.913,Y 82.697,Z 65.150,A 180.000,B 0.000,C 180.000} C_DIS
LIN {X 99.445,Y 82.631,Z 65.133,A 180.000,B 0.000,C 180.000} C_DIS
LIN {X 99.289,Y 82.609,Z 65.128,A 180.000,B 0.000,C 180.000} C_DIS
LIN {X 99.211,Y 82.598,Z 65.125,A 180.000,B 0.000,C 180.000} C_DIS
LIN {X 99.133,Y 82.589,Z 65.122,A 180.000,B 0.000,C 180.000} C_DIS
LIN {X 99.054,Y 82.583,Z 65.120,A 180.000,B 0.000,C 180.000} C_DIS
LIN {X 98.819,Y 82.563,Z 65.111,A 180.000,B 0.000,C 180.000} C_DIS
LIN {X 98.662,Y 82.550,Z 65.106,A 180.000,B 0.000,C 180.000} C_DIS
LIN {X 98.426,Y 82.530,Z 65.098,A 180.000,B 0.000,C 180.000} C_DIS
LIN {X 98.348,Y 82.524,Z 65.095,A 180.000,B 0.000,C 180.000} C_DIS
LIN {X 98.269,Y 82.521,Z 65.092,A 180.000,B 0.000,C 180.000} C_DIS
LIN {X 97.639,Y 82.503,Z 65.070,A 180.000,B 0.000,C 180.000} C_DIS
LIN {X 97.561,Y 82.501,Z 65.067,A 180.000,B 0.000,C 180.000} C_DIS
LIN {X 97.482,Y 82.500,Z 65.065,A 180.000,B 0.000,C 180.000} C_DIS
LIN {X 97.403,Y 82.502,Z 65.062,A 180.000,B 0.000,C 180.000} C_DIS
LIN {X 96.773,Y 82.519,Z 65.040,A 180.000,B 0.000,C 180.000} C_DIS
LIN {X 96.695,Y 82.522,Z 65.037,A 180.000,B 0.000,C 180.000} C_DIS
LIN {X 96.616,Y 82.526,Z 65.034,A 180.000,B 0.000,C 180.000} C_DIS
LIN {X 96.538,Y 82.533,Z 65.032,A 180.000,B 0.000,C 180.000} C_DIS
LIN {X 95.910,Y 82.586,Z 65.010,A 180.000,B 0.000,C 180.000} C_DIS
LIN {X 95.831,Y 82.593,Z 65.007,A 180.000,B 0.000,C 180.000} C_DIS
LIN {X 95.753,Y 82.603,Z 65.004,A 180.000,B 0.000,C 180.000} C_DIS
LIN {X 95.051,Y 82.702,Z 64.979,A 180.000,B 0.000,C 180.000} C_DIS
LIN {X 94.974,Y 82.714,Z 64.977,A 180.000,B 0.000,C 180.000} C_DIS
LIN {X 94.896,Y 82.729,Z 64.974,A 180.000,B 0.000,C 180.000} C_DIS
LIN {X 94.278,Y 82.852,Z 64.952,A 180.000,B 0.000,C 180.000} C_DIS
LIN {X 94.201,Y 82.868,Z 64.949,A 180.000,B 0.000,C 180.000} C_DIS
LIN {X 94.124,Y 82.885,Z 64.946,A 180.000,B 0.000,C 180.000} C_DIS
LIN {X 94.048,Y 82.904,Z 64.944,A 180.000,B 0.000,C 180.000} C_DIS
LIN {X 93.514,Y 83.042,Z 64.924,A 180.000,B 0.000,C 180.000} C_DIS
LIN {X 93.438,Y 83.062,Z 64.922,A 180.000,B 0.000,C 180.000} C_DIS
LIN {X 93.362,Y 83.082,Z 64.919,A 180.000,B 0.000,C 180.000} C_DIS
LIN {X 93.286,Y 83.105,Z 64.916,A 180.000,B 0.000,C 180.000} C_DIS
LIN {X 93.136,Y 83.152,Z 64.911,A 180.000,B 0.000,C 180.000} C_DIS
LIN {X 92.911,Y 83.224,Z 64.902,A 180.000,B 0.000,C 180.000} C_DIS
LIN {X 92.686,Y 83.296,Z 64.894,A 180.000,B 0.000,C 180.000} C_DIS
LIN {X 92.611,Y 83.320,Z 64.891,A 180.000,B 0.000,C 180.000} C_DIS
LIN {X 92.537,Y 83.345,Z 64.889,A 180.000,B 0.000,C 180.000} C_DIS
LIN {X 92.463,Y 83.372,Z 64.886,A 180.000,B 0.000,C 180.000} C_DIS
LIN {X 92.021,Y 83.541,Z 64.869,A 180.000,B 0.000,C 180.000} C_DIS
LIN {X 91.874,Y 83.597,Z 64.864,A 180.000,B 0.000,C 180.000} C_DIS
LIN {X 91.801,Y 83.625,Z 64.861,A 180.000,B 0.000,C 180.000} C_DIS
LIN {X 91.728,Y 83.655,Z 64.858,A 180.000,B 0.000,C 180.000} C_DIS
LIN {X 91.656,Y 83.687,Z 64.856,A 180.000,B 0.000,C 180.000} C_DIS
LIN {X 91.440,Y 83.784,Z 64.847,A 180.000,B 0.000,C 180.000} C_DIS
LIN {X 91.296,Y 83.848,Z 64.842,A 180.000,B 0.000,C 180.000} C_DIS
LIN {X 91.081,Y 83.945,Z 64.834,A 180.000,B 0.000,C 180.000} C_DIS
LIN {X 91.009,Y 83.977,Z 64.831,A 180.000,B 0.000,C 180.000} C_DIS
LIN {X 90.938,Y 84.012,Z 64.828,A 180.000,B 0.000,C 180.000} C_DIS
LIN {X 90.868,Y 84.048,Z 64.825,A 180.000,B 0.000,C 180.000} C_DIS
LIN {X 90.798,Y 84.084,Z 64.823,A 180.000,B 0.000,C 180.000} C_DIS
LIN {X 90.659,Y 84.156,Z 64.817,A 180.000,B 0.000,C 180.000} C_DIS
LIN {X 90.309,Y 84.337,Z 64.803,A 180.000,B 0.000,C 180.000} C_DIS
LIN {X 90.239,Y 84.374,Z 64.801,A 180.000,B 0.000,C 180.000} C_DIS
LIN {X 90.171,Y 84.414,Z 64.798,A 180.000,B 0.000,C 180.000} C_DIS
LIN {X 90.035,Y 84.494,Z 64.792,A 180.000,B 0.000,C 180.000} C_DIS
LIN {X 89.968,Y 84.534,Z 64.790,A 180.000,B 0.000,C 180.000} C_DIS
LIN {X 89.832,Y 84.614,Z 64.784,A 180.000,B 0.000,C 180.000} C_DIS
LIN {X 89.628,Y 84.734,Z 64.776,A 180.000,B 0.000,C 180.000} C_DIS
LIN {X 89.561,Y 84.774,Z 64.773,A 180.000,B 0.000,C 180.000} C_DIS
LIN {X 89.494,Y 84.816,Z 64.770,A 180.000,B 0.000,C 180.000} C_DIS
LIN {X 89.428,Y 84.859,Z 64.768,A 180.000,B 0.000,C 180.000} C_DIS
LIN {X 89.297,Y 84.947,Z 64.762,A 180.000,B 0.000,C 180.000} C_DIS
LIN {X 89.101,Y 85.078,Z 64.754,A 180.000,B 0.000,C 180.000} C_DIS
LIN {X 88.970,Y 85.165,Z 64.748,A 180.000,B 0.000,C 180.000} C_DIS
LIN {X 88.904,Y 85.209,Z 64.746,A 180.000,B 0.000,C 180.000} C_DIS
LIN {X 88.839,Y 85.253,Z 64.743,A 180.000,B 0.000,C 180.000} C_DIS
LIN {X 88.775,Y 85.299,Z 64.740,A 180.000,B 0.000,C 180.000} C_DIS
LIN {X 88.712,Y 85.346,Z 64.737,A 180.000,B 0.000,C 180.000} C_DIS
LIN {X 88.649,Y 85.394,Z 64.735,A 180.000,B 0.000,C 180.000} C_DIS
LIN {X 88.523,Y 85.488,Z 64.729,A 180.000,B 0.000,C 180.000} C_DIS
LIN {X 88.335,Y 85.631,Z 64.721,A 180.000,B 0.000,C 180.000} C_DIS
LIN {X 88.209,Y 85.725,Z 64.715,A 180.000,B 0.000,C 180.000} C_DIS
LIN {X 88.147,Y 85.773,Z 64.713,A 180.000,B 0.000,C 180.000} C_DIS
LIN {X 88.086,Y 85.824,Z 64.710,A 180.000,B 0.000,C 180.000} C_DIS
LIN {X 87.965,Y 85.925,Z 64.704,A 180.000,B 0.000,C 180.000} C_DIS
LIN {X 87.905,Y 85.976,Z 64.702,A 180.000,B 0.000,C 180.000} C_DIS
LIN {X 87.785,Y 86.078,Z 64.696,A 180.000,B 0.000,C 180.000} C_DIS
LIN {X 87.665,Y 86.179,Z 64.691,A 180.000,B 0.000,C 180.000} C_DIS
LIN {X 87.604,Y 86.230,Z 64.688,A 180.000,B 0.000,C 180.000} C_DIS
LIN {X 87.544,Y 86.281,Z 64.685,A 180.000,B 0.000,C 180.000} C_DIS
LIN {X 87.485,Y 86.333,Z 64.682,A 180.000,B 0.000,C 180.000} C_DIS
LIN {X 87.428,Y 86.387,Z 64.680,A 180.000,B 0.000,C 180.000} C_DIS
LIN {X 87.313,Y 86.495,Z 64.674,A 180.000,B 0.000,C 180.000} C_DIS
LIN {X 87.199,Y 86.603,Z 64.669,A 180.000,B 0.000,C 180.000} C_DIS
LIN {X 87.084,Y 86.711,Z 64.664,A 180.000,B 0.000,C 180.000} C_DIS
LIN {X 87.027,Y 86.766,Z 64.661,A 180.000,B 0.000,C 180.000} C_DIS
LIN {X 86.970,Y 86.820,Z 64.659,A 180.000,B 0.000,C 180.000} C_DIS
LIN {X 86.913,Y 86.874,Z 64.656,A 180.000,B 0.000,C 180.000} C_DIS
LIN {X 86.858,Y 86.930,Z 64.654,A 180.000,B 0.000,C 180.000} C_DIS
LIN {X 86.803,Y 86.987,Z 64.651,A 180.000,B 0.000,C 180.000} C_DIS
LIN {X 86.749,Y 87.044,Z 64.648,A 180.000,B 0.000,C 180.000} C_DIS
LIN {X 86.641,Y 87.159,Z 64.644,A 180.000,B 0.000,C 180.000} C_DIS
LIN {X 86.533,Y 87.273,Z 64.639,A 180.000,B 0.000,C 180.000} C_DIS
LIN {X 86.425,Y 87.388,Z 64.634,A 180.000,B 0.000,C 180.000} C_DIS
LIN {X 86.317,Y 87.503,Z 64.629,A 180.000,B 0.000,C 180.000} C_DIS
LIN {X 86.215,Y 87.622,Z 64.624,A 180.000,B 0.000,C 180.000} C_DIS
LIN {X 86.113,Y 87.743,Z 64.620,A 180.000,B 0.000,C 180.000} C_DIS
LIN {X 86.012,Y 87.863,Z 64.615,A 180.000,B 0.000,C 180.000} C_DIS
LIN {X 85.910,Y 87.983,Z 64.610,A 180.000,B 0.000,C 180.000} C_DIS
LIN {X 85.808,Y 88.104,Z 64.606,A 180.000,B 0.000,C 180.000} C_DIS
LIN {X 85.711,Y 88.228,Z 64.602,A 180.000,B 0.000,C 180.000} C_DIS
LIN {X 85.616,Y 88.353,Z 64.597,A 180.000,B 0.000,C 180.000} C_DIS
LIN {X 85.522,Y 88.479,Z 64.593,A 180.000,B 0.000,C 180.000} C_DIS
LIN {X 85.427,Y 88.605,Z 64.589,A 180.000,B 0.000,C 180.000} C_DIS
LIN {X 85.332,Y 88.731,Z 64.585,A 180.000,B 0.000,C 180.000} C_DIS
LIN {X 85.240,Y 88.858,Z 64.581,A 180.000,B 0.000,C 180.000} C_DIS
LIN {X 85.152,Y 88.989,Z 64.577,A 180.000,B 0.000,C 180.000} C_DIS
LIN {X 85.065,Y 89.120,Z 64.573,A 180.000,B 0.000,C 180.000} C_DIS
LIN {X 84.977,Y 89.251,Z 64.570,A 180.000,B 0.000,C 180.000} C_DIS
LIN {X 84.890,Y 89.382,Z 64.566,A 180.000,B 0.000,C 180.000} C_DIS
LIN {X 84.803,Y 89.514,Z 64.562,A 180.000,B 0.000,C 180.000} C_DIS
LIN {X 84.722,Y 89.649,Z 64.559,A 180.000,B 0.000,C 180.000} C_DIS
LIN {X 84.642,Y 89.784,Z 64.556,A 180.000,B 0.000,C 180.000} C_DIS
LIN {X 84.562,Y 89.920,Z 64.552,A 180.000,B 0.000,C 180.000} C_DIS
LIN {X 84.482,Y 90.056,Z 64.549,A 180.000,B 0.000,C 180.000} C_DIS
LIN {X 84.402,Y 90.191,Z 64.546,A 180.000,B 0.000,C 180.000} C_DIS
LIN {X 84.326,Y 90.330,Z 64.543,A 180.000,B 0.000,C 180.000} C_DIS
LIN {X 84.254,Y 90.470,Z 64.540,A 180.000,B 0.000,C 180.000} C_DIS
LIN {X 84.182,Y 90.610,Z 64.537,A 180.000,B 0.000,C 180.000} C_DIS
LIN {X 84.110,Y 90.749,Z 64.534,A 180.000,B 0.000,C 180.000} C_DIS
LIN {X 84.037,Y 90.889,Z 64.532,A 180.000,B 0.000,C 180.000} C_DIS
LIN {X 83.967,Y 91.030,Z 64.529,A 180.000,B 0.000,C 180.000} C_DIS
LIN {X 83.903,Y 91.174,Z 64.527,A 180.000,B 0.000,C 180.000} C_DIS
LIN {X 83.774,Y 91.462,Z 64.522,A 180.000,B 0.000,C 180.000} C_DIS
LIN {X 83.646,Y 91.749,Z 64.518,A 180.000,B 0.000,C 180.000} C_DIS
LIN {X 83.533,Y 92.043,Z 64.514,A 180.000,B 0.000,C 180.000} C_DIS
LIN {X 83.420,Y 92.338,Z 64.511,A 180.000,B 0.000,C 180.000} C_DIS
LIN {X 83.313,Y 92.634,Z 64.508,A 180.000,B 0.000,C 180.000} C_DIS
LIN {X 83.217,Y 92.934,Z 64.505,A 180.000,B 0.000,C 180.000} C_DIS
LIN {X 83.121,Y 93.234,Z 64.503,A 180.000,B 0.000,C 180.000} C_DIS
LIN {X 83.036,Y 93.537,Z 64.502,A 180.000,B 0.000,C 180.000} C_DIS
LIN {X 82.958,Y 93.842,Z 64.501,A 180.000,B 0.000,C 180.000} C_DIS
LIN {X 82.880,Y 94.147,Z 64.500,A 180.000,B 0.000,C 180.000} C_DIS
LIN {X 82.833,Y 94.374,Z 64.500,A 180.000,B 0.000,C 180.000} C_DIS
; Cutting Move Starts
LIN {X 82.829,Y 94.394,Z 64.500,A 180.000,B 0.000,C 180.000} C_DIS
LIN {X 82.758,Y 94.751,Z 64.500,A 180.000,B 0.000,C 180.000} C_DIS
LIN {X 82.722,Y 94.930,Z 64.500,A 180.000,B 0.000,C 180.000} C_DIS
LIN {X 82.694,Y 95.109,Z 64.500,A 180.000,B 0.000,C 180.000} C_DIS
LIN {X 82.618,Y 95.645,Z 64.500,A 180.000,B 0.000,C 180.000} C_DIS
LIN {X 82.595,Y 95.815,Z 64.500,A 180.000,B 0.000,C 180.000} C_DIS
LIN {X 82.594,Y 95.824,Z 64.500,A 180.000,B 0.000,C 180.000} C_DIS
LIN {X 82.578,Y 96.003,Z 64.500,A 180.000,B 0.000,C 180.000} C_DIS
LIN {X 82.533,Y 96.539,Z 64.500,A 180.000,B 0.000,C 180.000} C_DIS
LIN {X 82.521,Y 96.718,Z 64.500,A 180.000,B 0.000,C 180.000} C_DIS
LIN {X 82.516,Y 96.897,Z 64.500,A 180.000,B 0.000,C 180.000} C_DIS
LIN {X 82.501,Y 97.433,Z 64.500,A 180.000,B 0.000,C 180.000} C_DIS
LIN {X 82.502,Y 97.612,Z 64.500,A 180.000,B 0.000,C 180.000} C_DIS
LIN {X 82.517,Y 98.148,Z 64.500,A 180.000,B 0.000,C 180.000} C_DIS
LIN {X 82.523,Y 98.327,Z 64.500,A 180.000,B 0.000,C 180.000} C_DIS
LIN {X 82.536,Y 98.505,Z 64.500,A 180.000,B 0.000,C 180.000} C_DIS
LIN {X 82.582,Y 99.042,Z 64.500,A 180.000,B 0.000,C 180.000} C_DIS
LIN {X 82.595,Y 99.185,Z 64.500,A 180.000,B 0.000,C 180.000} C_DIS
LIN {X 82.599,Y 99.221,Z 64.500,A 180.000,B 0.000,C 180.000} C_DIS
LIN {X 82.624,Y 99.399,Z 64.500,A 180.000,B 0.000,C 180.000} C_DIS
LIN {X 82.700,Y 99.936,Z 64.500,A 180.000,B 0.000,C 180.000} C_DIS
LIN {X 82.731,Y 100.114,Z 64.500,A 180.000,B 0.000,C 180.000} C_DIS
LIN {X 82.838,Y 100.651,Z 64.500,A 180.000,B 0.000,C 180.000} C_DIS
LIN {X 82.874,Y 100.829,Z 64.500,A 180.000,B 0.000,C 180.000} C_DIS
LIN {X 82.919,Y 101.008,Z 64.500,A 180.000,B 0.000,C 180.000} C_DIS
LIN {X 83.057,Y 101.545,Z 64.500,A 180.000,B 0.000,C 180.000} C_DIS
LIN {X 83.108,Y 101.723,Z 64.500,A 180.000,B 0.000,C 180.000} C_DIS
LIN {X 83.310,Y 102.358,Z 64.500,A 180.000,B 0.000,C 180.000} C_DIS
LIN {X 83.336,Y 102.438,Z 64.500,A 180.000,B 0.000,C 180.000} C_DIS
LIN {X 83.403,Y 102.617,Z 64.500,A 180.000,B 0.000,C 180.000} C_DIS
LIN {X 83.608,Y 103.153,Z 64.500,A 180.000,B 0.000,C 180.000} C_DIS
LIN {X 83.668,Y 103.300,Z 64.500,A 180.000,B 0.000,C 180.000} C_DIS
LIN {X 83.922,Y 103.869,Z 64.500,A 180.000,B 0.000,C 180.000} C_DIS
LIN {X 84.005,Y 104.047,Z 64.500,A 180.000,B 0.000,C 180.000} C_DIS
LIN {X 84.025,Y 104.087,Z 64.500,A 180.000,B 0.000,C 180.000} C_DIS
LIN {X 84.282,Y 104.584,Z 64.500,A 180.000,B 0.000,C 180.000} C_DIS
LIN {X 84.375,Y 104.762,Z 64.500,A 180.000,B 0.000,C 180.000} C_DIS
LIN {X 84.383,Y 104.775,Z 64.500,A 180.000,B 0.000,C 180.000} C_DIS
LIN {X 84.480,Y 104.941,Z 64.500,A 180.000,B 0.000,C 180.000} C_DIS
LIN {X 84.740,Y 105.382,Z 64.500,A 180.000,B 0.000,C 180.000} C_DIS
LIN {X 84.797,Y 105.477,Z 64.500,A 180.000,B 0.000,C 180.000} C_DIS
LIN {X 84.915,Y 105.656,Z 64.500,A 180.000,B 0.000,C 180.000} C_DIS
LIN {X 85.154,Y 106.014,Z 64.500,A 180.000,B 0.000,C 180.000} C_DIS
LIN {X 85.276,Y 106.193,Z 64.500,A 180.000,B 0.000,C 180.000} C_DIS
LIN {X 85.276,Y 106.194,Z 64.500,A 180.000,B 0.000,C 180.000} C_DIS
LIN {X 85.409,Y 106.371,Z 64.500,A 180.000,B 0.000,C 180.000} C_DIS
LIN {X 85.678,Y 106.729,Z 64.500,A 180.000,B 0.000,C 180.000} C_DIS
LIN {X 85.813,Y 106.902,Z 64.500,A 180.000,B 0.000,C 180.000} C_DIS
LIN {X 85.818,Y 106.908,Z 64.500,A 180.000,B 0.000,C 180.000} C_DIS
LIN {X 86.271,Y 107.444,Z 64.500,A 180.000,B 0.000,C 180.000} C_DIS
LIN {X 86.349,Y 107.532,Z 64.500,A 180.000,B 0.000,C 180.000} C_DIS
LIN {X 86.435,Y 107.623,Z 64.500,A 180.000,B 0.000,C 180.000} C_DIS
LIN {X 86.773,Y 107.980,Z 64.500,A 180.000,B 0.000,C 180.000} C_DIS
LIN {X 86.885,Y 108.099,Z 64.500,A 180.000,B 0.000,C 180.000} C_DIS
LIN {X 86.947,Y 108.159,Z 64.500,A 180.000,B 0.000,C 180.000} C_DIS
LIN {X 87.422,Y 108.607,Z 64.500,A 180.000,B 0.000,C 180.000} C_DIS
LIN {X 87.517,Y 108.695,Z 64.500,A 180.000,B 0.000,C 180.000} C_DIS
LIN {X 87.601,Y 108.767,Z 64.500,A 180.000,B 0.000,C 180.000} C_DIS
LIN {X 87.958,Y 109.069,Z 64.500,A 180.000,B 0.000,C 180.000} C_DIS
LIN {X 88.137,Y 109.219,Z 64.500,A 180.000,B 0.000,C 180.000} C_DIS
LIN {X 88.153,Y 109.232,Z 64.500,A 180.000,B 0.000,C 180.000} C_DIS
LIN {X 88.316,Y 109.355,Z 64.500,A 180.000,B 0.000,C 180.000} C_DIS
LIN {X 88.673,Y 109.624,Z 64.500,A 180.000,B 0.000,C 180.000} C_DIS
LIN {X 88.852,Y 109.756,Z 64.500,A 180.000,B 0.000,C 180.000} C_DIS
LIN {X 88.870,Y 109.768,Z 64.500,A 180.000,B 0.000,C 180.000} C_DIS
LIN {X 89.031,Y 109.875,Z 64.500,A 180.000,B 0.000,C 180.000} C_DIS
LIN {X 89.405,Y 110.126,Z 64.500,A 180.000,B 0.000,C 180.000} C_DIS
LIN {X 89.567,Y 110.230,Z 64.500,A 180.000,B 0.000,C 180.000} C_DIS
LIN {X 89.693,Y 110.304,Z 64.500,A 180.000,B 0.000,C 180.000} C_DIS
LIN {X 90.103,Y 110.546,Z 64.500,A 180.000,B 0.000,C 180.000} C_DIS
LIN {X 90.282,Y 110.649,Z 64.500,A 180.000,B 0.000,C 180.000} C_DIS
LIN {X 90.307,Y 110.662,Z 64.500,A 180.000,B 0.000,C 180.000} C_DIS
LIN {X 90.818,Y 110.926,Z 64.500,A 180.000,B 0.000,C 180.000} C_DIS
LIN {X 90.997,Y 111.017,Z 64.500,A 180.000,B 0.000,C 180.000} C_DIS
LIN {X 91.002,Y 111.019,Z 64.500,A 180.000,B 0.000,C 180.000} C_DIS
LIN {X 91.176,Y 111.098,Z 64.500,A 180.000,B 0.000,C 180.000} C_DIS
LIN {X 91.533,Y 111.258,Z 64.500,A 180.000,B 0.000,C 180.000} C_DIS
LIN {X 91.712,Y 111.338,Z 64.500,A 180.000,B 0.000,C 180.000} C_DIS
LIN {X 91.806,Y 111.377,Z 64.500,A 180.000,B 0.000,C 180.000} C_DIS
LIN {X 91.891,Y 111.409,Z 64.500,A 180.000,B 0.000,C 180.000} C_DIS
LIN {X 92.427,Y 111.614,Z 64.500,A 180.000,B 0.000,C 180.000} C_DIS
LIN {X 92.606,Y 111.678,Z 64.500,A 180.000,B 0.000,C 180.000} C_DIS
LIN {X 92.964,Y 111.792,Z 64.500,A 180.000,B 0.000,C 180.000} C_DIS
LIN {X 93.142,Y 111.849,Z 64.500,A 180.000,B 0.000,C 180.000} C_DIS
LIN {X 93.321,Y 111.906,Z 64.500,A 180.000,B 0.000,C 180.000} C_DIS
LIN {X 93.346,Y 111.913,Z 64.500,A 180.000,B 0.000,C 180.000} C_DIS
LIN {X 93.500,Y 111.954,Z 64.500,A 180.000,B 0.000,C 180.000} C_DIS
LIN {X 94.036,Y 112.092,Z 64.500,A 180.000,B 0.000,C 180.000} C_DIS
LIN {X 94.215,Y 112.135,Z 64.500,A 180.000,B 0.000,C 180.000} C_DIS
LIN {X 94.394,Y 112.171,Z 64.500,A 180.000,B 0.000,C 180.000} C_DIS
LIN {X 94.895,Y 112.271,Z 64.500,A 180.000,B 0.000,C 180.000} C_DIS
LIN {X 94.930,Y 112.278,Z 64.500,A 180.000,B 0.000,C 180.000} C_DIS
LIN {X 95.109,Y 112.306,Z 64.500,A 180.000,B 0.000,C 180.000} C_DIS
LIN {X 95.645,Y 112.382,Z 64.500,A 180.000,B 0.000,C 180.000} C_DIS
LIN {X 95.824,Y 112.406,Z 64.500,A 180.000,B 0.000,C 180.000} C_DIS
LIN {X 96.003,Y 112.422,Z 64.500,A 180.000,B 0.000,C 180.000} C_DIS
LIN {X 96.539,Y 112.467,Z 64.500,A 180.000,B 0.000,C 180.000} C_DIS
LIN {X 96.718,Y 112.479,Z 64.500,A 180.000,B 0.000,C 180.000} C_DIS
LIN {X 96.897,Y 112.484,Z 64.500,A 180.000,B 0.000,C 180.000} C_DIS
LIN {X 97.433,Y 112.499,Z 64.500,A 180.000,B 0.000,C 180.000} C_DIS
LIN {X 97.612,Y 112.498,Z 64.500,A 180.000,B 0.000,C 180.000} C_DIS
LIN {X 98.148,Y 112.483,Z 64.500,A 180.000,B 0.000,C 180.000} C_DIS
LIN {X 98.327,Y 112.477,Z 64.500,A 180.000,B 0.000,C 180.000} C_DIS
LIN {X 98.505,Y 112.464,Z 64.500,A 180.000,B 0.000,C 180.000} C_DIS
LIN {X 99.042,Y 112.418,Z 64.500,A 180.000,B 0.000,C 180.000} C_DIS
LIN {X 99.221,Y 112.401,Z 64.500,A 180.000,B 0.000,C 180.000} C_DIS
LIN {X 99.399,Y 112.376,Z 64.500,A 180.000,B 0.000,C 180.000} C_DIS
LIN {X 99.936,Y 112.300,Z 64.500,A 180.000,B 0.000,C 180.000} C_DIS
LIN {X 100.105,Y 112.271,Z 64.500,A 180.000,B 0.000,C 180.000} C_DIS
LIN {X 100.651,Y 112.162,Z 64.500,A 180.000,B 0.000,C 180.000} C_DIS
LIN {X 100.829,Y 112.126,Z 64.500,A 180.000,B 0.000,C 180.000} C_DIS
LIN {X 100.966,Y 112.092,Z 64.500,A 180.000,B 0.000,C 180.000} C_DIS
LIN {X 101.545,Y 111.943,Z 64.500,A 180.000,B 0.000,C 180.000} C_DIS
LIN {X 101.654,Y 111.913,Z 64.500,A 180.000,B 0.000,C 180.000} C_DIS
LIN {X 101.723,Y 111.892,Z 64.500,A 180.000,B 0.000,C 180.000} C_DIS
LIN {X 102.260,Y 111.721,Z 64.500,A 180.000,B 0.000,C 180.000} C_DIS
LIN {X 102.438,Y 111.664,Z 64.500,A 180.000,B 0.000,C 180.000} C_DIS
LIN {X 102.617,Y 111.597,Z 64.500,A 180.000,B 0.000,C 180.000} C_DIS
LIN {X 103.153,Y 111.392,Z 64.500,A 180.000,B 0.000,C 180.000} C_DIS
LIN {X 103.194,Y 111.377,Z 64.500,A 180.000,B 0.000,C 180.000} C_DIS
LIN {X 103.332,Y 111.318,Z 64.500,A 180.000,B 0.000,C 180.000} C_DIS
LIN {X 103.869,Y 111.078,Z 64.500,A 180.000,B 0.000,C 180.000} C_DIS
LIN {X 103.998,Y 111.019,Z 64.500,A 180.000,B 0.000,C 180.000} C_DIS
LIN {X 104.047,Y 110.995,Z 64.500,A 180.000,B 0.000,C 180.000} C_DIS
LIN {X 104.226,Y 110.903,Z 64.500,A 180.000,B 0.000,C 180.000} C_DIS
LIN {X 104.693,Y 110.662,Z 64.500,A 180.000,B 0.000,C 180.000} C_DIS
LIN {X 104.762,Y 110.625,Z 64.500,A 180.000,B 0.000,C 180.000} C_DIS
LIN {X 104.941,Y 110.520,Z 64.500,A 180.000,B 0.000,C 180.000} C_DIS
LIN {X 105.307,Y 110.304,Z 64.500,A 180.000,B 0.000,C 180.000} C_DIS
LIN {X 105.477,Y 110.203,Z 64.500,A 180.000,B 0.000,C 180.000} C_DIS
LIN {X 105.595,Y 110.126,Z 64.500,A 180.000,B 0.000,C 180.000} C_DIS
LIN {X 106.014,Y 109.846,Z 64.500,A 180.000,B 0.000,C 180.000} C_DIS
LIN {X 106.130,Y 109.768,Z 64.500,A 180.000,B 0.000,C 180.000} C_DIS
LIN {X 106.193,Y 109.724,Z 64.500,A 180.000,B 0.000,C 180.000} C_DIS
LIN {X 106.371,Y 109.591,Z 64.500,A 180.000,B 0.000,C 180.000} C_DIS
LIN {X 106.729,Y 109.322,Z 64.500,A 180.000,B 0.000,C 180.000} C_DIS
LIN {X 106.847,Y 109.232,Z 64.500,A 180.000,B 0.000,C 180.000} C_DIS
LIN {X 106.908,Y 109.182,Z 64.500,A 180.000,B 0.000,C 180.000} C_DIS
LIN {X 107.444,Y 108.729,Z 64.500,A 180.000,B 0.000,C 180.000} C_DIS
LIN {X 107.483,Y 108.695,Z 64.500,A 180.000,B 0.000,C 180.000} C_DIS
LIN {X 107.623,Y 108.565,Z 64.500,A 180.000,B 0.000,C 180.000} C_DIS
LIN {X 108.053,Y 108.159,Z 64.500,A 180.000,B 0.000,C 180.000} C_DIS
LIN {X 108.159,Y 108.053,Z 64.500,A 180.000,B 0.000,C 180.000} C_DIS
LIN {X 108.565,Y 107.623,Z 64.500,A 180.000,B 0.000,C 180.000} C_DIS
LIN {X 108.695,Y 107.483,Z 64.500,A 180.000,B 0.000,C 180.000} C_DIS
LIN {X 108.729,Y 107.444,Z 64.500,A 180.000,B 0.000,C 180.000} C_DIS
LIN {X 109.182,Y 106.908,Z 64.500,A 180.000,B 0.000,C 180.000} C_DIS
LIN {X 109.232,Y 106.847,Z 64.500,A 180.000,B 0.000,C 180.000} C_DIS
LIN {X 109.322,Y 106.729,Z 64.500,A 180.000,B 0.000,C 180.000} C_DIS
LIN {X 109.591,Y 106.371,Z 64.500,A 180.000,B 0.000,C 180.000} C_DIS
LIN {X 109.724,Y 106.193,Z 64.500,A 180.000,B 0.000,C 180.000} C_DIS
LIN {X 109.768,Y 106.130,Z 64.500,A 180.000,B 0.000,C 180.000} C_DIS
LIN {X 109.846,Y 106.014,Z 64.500,A 180.000,B 0.000,C 180.000} C_DIS
LIN {X 110.126,Y 105.595,Z 64.500,A 180.000,B 0.000,C 180.000} C_DIS
LIN {X 110.203,Y 105.477,Z 64.500,A 180.000,B 0.000,C 180.000} C_DIS
LIN {X 110.304,Y 105.307,Z 64.500,A 180.000,B 0.000,C 180.000} C_DIS
LIN {X 110.520,Y 104.941,Z 64.500,A 180.000,B 0.000,C 180.000} C_DIS
LIN {X 110.625,Y 104.762,Z 64.500,A 180.000,B 0.000,C 180.000} C_DIS
LIN {X 110.662,Y 104.693,Z 64.500,A 180.000,B 0.000,C 180.000} C_DIS
LIN {X 110.903,Y 104.226,Z 64.500,A 180.000,B 0.000,C 180.000} C_DIS
LIN {X 110.995,Y 104.047,Z 64.500,A 180.000,B 0.000,C 180.000} C_DIS
LIN {X 111.019,Y 103.998,Z 64.500,A 180.000,B 0.000,C 180.000} C_DIS
LIN {X 111.078,Y 103.869,Z 64.500,A 180.000,B 0.000,C 180.000} C_DIS
LIN {X 111.318,Y 103.332,Z 64.500,A 180.000,B 0.000,C 180.000} C_DIS
LIN {X 111.377,Y 103.194,Z 64.500,A 180.000,B 0.000,C 180.000} C_DIS
LIN {X 111.392,Y 103.153,Z 64.500,A 180.000,B 0.000,C 180.000} C_DIS
LIN {X 111.597,Y 102.617,Z 64.500,A 180.000,B 0.000,C 180.000} C_DIS
LIN {X 111.664,Y 102.438,Z 64.500,A 180.000,B 0.000,C 180.000} C_DIS
LIN {X 111.721,Y 102.260,Z 64.500,A 180.000,B 0.000,C 180.000} C_DIS
LIN {X 111.892,Y 101.723,Z 64.500,A 180.000,B 0.000,C 180.000} C_DIS
LIN {X 111.913,Y 101.654,Z 64.500,A 180.000,B 0.000,C 180.000} C_DIS
LIN {X 111.943,Y 101.545,Z 64.500,A 180.000,B 0.000,C 180.000} C_DIS
LIN {X 112.092,Y 100.966,Z 64.500,A 180.000,B 0.000,C 180.000} C_DIS
LIN {X 112.126,Y 100.829,Z 64.500,A 180.000,B 0.000,C 180.000} C_DIS
LIN {X 112.162,Y 100.651,Z 64.500,A 180.000,B 0.000,C 180.000} C_DIS
LIN {X 112.271,Y 100.105,Z 64.500,A 180.000,B 0.000,C 180.000} C_DIS
LIN {X 112.300,Y 99.936,Z 64.500,A 180.000,B 0.000,C 180.000} C_DIS
LIN {X 112.376,Y 99.399,Z 64.500,A 180.000,B 0.000,C 180.000} C_DIS
LIN {X 112.401,Y 99.221,Z 64.500,A 180.000,B 0.000,C 180.000} C_DIS
LIN {X 112.418,Y 99.042,Z 64.500,A 180.000,B 0.000,C 180.000} C_DIS
LIN {X 112.464,Y 98.505,Z 64.500,A 180.000,B 0.000,C 180.000} C_DIS
LIN {X 112.477,Y 98.327,Z 64.500,A 180.000,B 0.000,C 180.000} C_DIS
LIN {X 112.483,Y 98.148,Z 64.500,A 180.000,B 0.000,C 180.000} C_DIS
LIN {X 112.498,Y 97.612,Z 64.500,A 180.000,B 0.000,C 180.000} C_DIS
LIN {X 112.499,Y 97.433,Z 64.500,A 180.000,B 0.000,C 180.000} C_DIS
LIN {X 112.484,Y 96.897,Z 64.500,A 180.000,B 0.000,C 180.000} C_DIS
LIN {X 112.479,Y 96.718,Z 64.500,A 180.000,B 0.000,C 180.000} C_DIS
LIN {X 112.467,Y 96.539,Z 64.500,A 180.000,B 0.000,C 180.000} C_DIS
LIN {X 112.422,Y 96.003,Z 64.500,A 180.000,B 0.000,C 180.000} C_DIS
LIN {X 112.406,Y 95.824,Z 64.500,A 180.000,B 0.000,C 180.000} C_DIS
LIN {X 112.382,Y 95.645,Z 64.500,A 180.000,B 0.000,C 180.000} C_DIS
LIN {X 112.306,Y 95.109,Z 64.500,A 180.000,B 0.000,C 180.000} C_DIS
LIN {X 112.278,Y 94.930,Z 64.500,A 180.000,B 0.000,C 180.000} C_DIS
LIN {X 112.271,Y 94.895,Z 64.500,A 180.000,B 0.000,C 180.000} C_DIS
LIN {X 112.171,Y 94.394,Z 64.500,A 180.000,B 0.000,C 180.000} C_DIS
LIN {X 112.135,Y 94.215,Z 64.500,A 180.000,B 0.000,C 180.000} C_DIS
LIN {X 112.092,Y 94.036,Z 64.500,A 180.000,B 0.000,C 180.000} C_DIS
LIN {X 111.954,Y 93.500,Z 64.500,A 180.000,B 0.000,C 180.000} C_DIS
LIN {X 111.913,Y 93.346,Z 64.500,A 180.000,B 0.000,C 180.000} C_DIS
LIN {X 111.906,Y 93.321,Z 64.500,A 180.000,B 0.000,C 180.000} C_DIS
LIN {X 111.849,Y 93.142,Z 64.500,A 180.000,B 0.000,C 180.000} C_DIS
LIN {X 111.734,Y 92.782,Z 64.500,A 180.000,B 0.000,C 180.000} C_DIS
LIN {X 111.678,Y 92.606,Z 64.500,A 180.000,B 0.000,C 180.000} C_DIS
LIN {X 111.614,Y 92.427,Z 64.500,A 180.000,B 0.000,C 180.000} C_DIS
LIN {X 111.409,Y 91.891,Z 64.500,A 180.000,B 0.000,C 180.000} C_DIS
LIN {X 111.377,Y 91.806,Z 64.500,A 180.000,B 0.000,C 180.000} C_DIS
LIN {X 111.338,Y 91.712,Z 64.500,A 180.000,B 0.000,C 180.000} C_DIS
LIN {X 111.258,Y 91.533,Z 64.500,A 180.000,B 0.000,C 180.000} C_DIS
LIN {X 111.098,Y 91.176,Z 64.500,A 180.000,B 0.000,C 180.000} C_DIS
LIN {X 111.019,Y 91.002,Z 64.500,A 180.000,B 0.000,C 180.000} C_DIS
LIN {X 111.017,Y 90.997,Z 64.500,A 180.000,B 0.000,C 180.000} C_DIS
LIN {X 110.946,Y 90.857,Z 64.500,A 180.000,B 0.000,C 180.000} C_DIS
LIN {X 110.926,Y 90.818,Z 64.500,A 180.000,B 0.000,C 180.000} C_DIS
LIN {X 110.662,Y 90.307,Z 64.500,A 180.000,B 0.000,C 180.000} C_DIS
LIN {X 110.649,Y 90.282,Z 64.500,A 180.000,B 0.000,C 180.000} C_DIS
LIN {X 110.546,Y 90.103,Z 64.500,A 180.000,B 0.000,C 180.000} C_DIS
LIN {X 110.304,Y 89.693,Z 64.500,A 180.000,B 0.000,C 180.000} C_DIS
LIN {X 110.230,Y 89.567,Z 64.500,A 180.000,B 0.000,C 180.000} C_DIS
LIN {X 110.126,Y 89.405,Z 64.500,A 180.000,B 0.000,C 180.000} C_DIS
LIN {X 109.875,Y 89.031,Z 64.500,A 180.000,B 0.000,C 180.000} C_DIS
LIN {X 109.768,Y 88.870,Z 64.500,A 180.000,B 0.000,C 180.000} C_DIS
LIN {X 109.756,Y 88.852,Z 64.500,A 180.000,B 0.000,C 180.000} C_DIS
LIN {X 109.624,Y 88.673,Z 64.500,A 180.000,B 0.000,C 180.000} C_DIS
LIN {X 109.355,Y 88.316,Z 64.500,A 180.000,B 0.000,C 180.000} C_DIS
LIN {X 109.232,Y 88.153,Z 64.500,A 180.000,B 0.000,C 180.000} C_DIS
LIN {X 109.219,Y 88.137,Z 64.500,A 180.000,B 0.000,C 180.000} C_DIS
LIN {X 109.069,Y 87.958,Z 64.500,A 180.000,B 0.000,C 180.000} C_DIS
LIN {X 108.767,Y 87.601,Z 64.500,A 180.000,B 0.000,C 180.000} C_DIS
LIN {X 108.695,Y 87.517,Z 64.500,A 180.000,B 0.000,C 180.000} C_DIS
LIN {X 108.607,Y 87.422,Z 64.500,A 180.000,B 0.000,C 180.000} C_DIS
LIN {X 108.159,Y 86.947,Z 64.500,A 180.000,B 0.000,C 180.000} C_DIS
LIN {X 108.099,Y 86.885,Z 64.500,A 180.000,B 0.000,C 180.000} C_DIS
LIN {X 107.980,Y 86.773,Z 64.500,A 180.000,B 0.000,C 180.000} C_DIS
LIN {X 107.623,Y 86.435,Z 64.500,A 180.000,B 0.000,C 180.000} C_DIS
LIN {X 107.532,Y 86.349,Z 64.500,A 180.000,B 0.000,C 180.000} C_DIS
LIN {X 107.444,Y 86.271,Z 64.500,A 180.000,B 0.000,C 180.000} C_DIS
LIN {X 106.908,Y 85.818,Z 64.500,A 180.000,B 0.000,C 180.000} C_DIS
LIN {X 106.902,Y 85.813,Z 64.500,A 180.000,B 0.000,C 180.000} C_DIS
LIN {X 106.729,Y 85.678,Z 64.500,A 180.000,B 0.000,C 180.000} C_DIS
LIN {X 106.371,Y 85.409,Z 64.500,A 180.000,B 0.000,C 180.000} C_DIS
LIN {X 106.194,Y 85.276,Z 64.500,A 180.000,B 0.000,C 180.000} C_DIS
LIN {X 106.193,Y 85.276,Z 64.500,A 180.000,B 0.000,C 180.000} C_DIS
LIN {X 106.014,Y 85.154,Z 64.500,A 180.000,B 0.000,C 180.000} C_DIS
LIN {X 105.656,Y 84.915,Z 64.500,A 180.000,B 0.000,C 180.000} C_DIS
LIN {X 105.477,Y 84.797,Z 64.500,A 180.000,B 0.000,C 180.000} C_DIS
LIN {X 105.382,Y 84.740,Z 64.500,A 180.000,B 0.000,C 180.000} C_DIS
LIN {X 104.941,Y 84.480,Z 64.500,A 180.000,B 0.000,C 180.000} C_DIS
LIN {X 104.775,Y 84.383,Z 64.500,A 180.000,B 0.000,C 180.000} C_DIS
LIN {X 104.762,Y 84.375,Z 64.500,A 180.000,B 0.000,C 180.000} C_DIS
LIN {X 104.584,Y 84.282,Z 64.500,A 180.000,B 0.000,C 180.000} C_DIS
LIN {X 104.087,Y 84.025,Z 64.500,A 180.000,B 0.000,C 180.000} C_DIS
LIN {X 104.047,Y 84.005,Z 64.500,A 180.000,B 0.000,C 180.000} C_DIS
LIN {X 103.869,Y 83.922,Z 64.500,A 180.000,B 0.000,C 180.000} C_DIS
LIN {X 103.300,Y 83.668,Z 64.500,A 180.000,B 0.000,C 180.000} C_DIS
LIN {X 103.153,Y 83.608,Z 64.500,A 180.000,B 0.000,C 180.000} C_DIS
LIN {X 102.617,Y 83.403,Z 64.500,A 180.000,B 0.000,C 180.000} C_DIS
LIN {X 102.438,Y 83.336,Z 64.500,A 180.000,B 0.000,C 180.000} C_DIS
LIN {X 102.358,Y 83.310,Z 64.500,A 180.000,B 0.000,C 180.000} C_DIS
LIN {X 101.723,Y 83.108,Z 64.500,A 180.000,B 0.000,C 180.000} C_DIS
LIN {X 101.545,Y 83.057,Z 64.500,A 180.000,B 0.000,C 180.000} C_DIS
LIN {X 101.008,Y 82.919,Z 64.500,A 180.000,B 0.000,C 180.000} C_DIS
LIN {X 100.829,Y 82.874,Z 64.500,A 180.000,B 0.000,C 180.000} C_DIS
LIN {X 100.651,Y 82.838,Z 64.500,A 180.000,B 0.000,C 180.000} C_DIS
LIN {X 100.114,Y 82.731,Z 64.500,A 180.000,B 0.000,C 180.000} C_DIS
LIN {X 99.936,Y 82.700,Z 64.500,A 180.000,B 0.000,C 180.000} C_DIS
LIN {X 99.399,Y 82.624,Z 64.500,A 180.000,B 0.000,C 180.000} C_DIS
LIN {X 99.221,Y 82.599,Z 64.500,A 180.000,B 0.000,C 180.000} C_DIS
LIN {X 99.185,Y 82.595,Z 64.500,A 180.000,B 0.000,C 180.000} C_DIS
LIN {X 99.042,Y 82.582,Z 64.500,A 180.000,B 0.000,C 180.000} C_DIS
LIN {X 98.505,Y 82.536,Z 64.500,A 180.000,B 0.000,C 180.000} C_DIS
LIN {X 98.327,Y 82.523,Z 64.500,A 180.000,B 0.000,C 180.000} C_DIS
LIN {X 98.148,Y 82.517,Z 64.500,A 180.000,B 0.000,C 180.000} C_DIS
LIN {X 97.612,Y 82.502,Z 64.500,A 180.000,B 0.000,C 180.000} C_DIS
LIN {X 97.433,Y 82.501,Z 64.500,A 180.000,B 0.000,C 180.000} C_DIS
LIN {X 96.897,Y 82.516,Z 64.500,A 180.000,B 0.000,C 180.000} C_DIS
LIN {X 96.718,Y 82.521,Z 64.500,A 180.000,B 0.000,C 180.000} C_DIS
LIN {X 96.539,Y 82.533,Z 64.500,A 180.000,B 0.000,C 180.000} C_DIS
LIN {X 96.003,Y 82.578,Z 64.500,A 180.000,B 0.000,C 180.000} C_DIS
LIN {X 95.824,Y 82.594,Z 64.500,A 180.000,B 0.000,C 180.000} C_DIS
LIN {X 95.815,Y 82.595,Z 64.500,A 180.000,B 0.000,C 180.000} C_DIS
LIN {X 95.645,Y 82.618,Z 64.500,A 180.000,B 0.000,C 180.000} C_DIS
LIN {X 95.109,Y 82.694,Z 64.500,A 180.000,B 0.000,C 180.000} C_DIS
LIN {X 94.930,Y 82.722,Z 64.500,A 180.000,B 0.000,C 180.000} C_DIS
LIN {X 94.751,Y 82.758,Z 64.500,A 180.000,B 0.000,C 180.000} C_DIS
LIN {X 94.394,Y 82.829,Z 64.500,A 180.000,B 0.000,C 180.000} C_DIS
LIN {X 94.215,Y 82.865,Z 64.500,A 180.000,B 0.000,C 180.000} C_DIS
LIN {X 94.036,Y 82.908,Z 64.500,A 180.000,B 0.000,C 180.000} C_DIS
LIN {X 93.500,Y 83.046,Z 64.500,A 180.000,B 0.000,C 180.000} C_DIS
LIN {X 93.321,Y 83.094,Z 64.500,A 180.000,B 0.000,C 180.000} C_DIS
LIN {X 93.203,Y 83.131,Z 64.500,A 180.000,B 0.000,C 180.000} C_DIS
LIN {X 92.642,Y 83.310,Z 64.500,A 180.000,B 0.000,C 180.000} C_DIS
LIN {X 92.606,Y 83.322,Z 64.500,A 180.000,B 0.000,C 180.000} C_DIS
LIN {X 92.427,Y 83.386,Z 64.500,A 180.000,B 0.000,C 180.000} C_DIS
LIN {X 91.891,Y 83.591,Z 64.500,A 180.000,B 0.000,C 180.000} C_DIS
LIN {X 91.712,Y 83.662,Z 64.500,A 180.000,B 0.000,C 180.000} C_DIS
LIN {X 91.700,Y 83.668,Z 64.500,A 180.000,B 0.000,C 180.000} C_DIS
LIN {X 91.176,Y 83.902,Z 64.500,A 180.000,B 0.000,C 180.000} C_DIS
LIN {X 90.997,Y 83.983,Z 64.500,A 180.000,B 0.000,C 180.000} C_DIS
LIN {X 90.913,Y 84.025,Z 64.500,A 180.000,B 0.000,C 180.000} C_DIS
LIN {X 90.461,Y 84.259,Z 64.500,A 180.000,B 0.000,C 180.000} C_DIS
LIN {X 90.282,Y 84.351,Z 64.500,A 180.000,B 0.000,C 180.000} C_DIS
LIN {X 90.225,Y 84.383,Z 64.500,A 180.000,B 0.000,C 180.000} C_DIS
LIN {X 90.103,Y 84.454,Z 64.500,A 180.000,B 0.000,C 180.000} C_DIS
LIN {X 89.618,Y 84.740,Z 64.500,A 180.000,B 0.000,C 180.000} C_DIS
LIN {X 89.567,Y 84.770,Z 64.500,A 180.000,B 0.000,C 180.000} C_DIS
LIN {X 89.388,Y 84.886,Z 64.500,A 180.000,B 0.000,C 180.000} C_DIS
LIN {X 89.031,Y 85.125,Z 64.500,A 180.000,B 0.000,C 180.000} C_DIS
LIN {X 88.852,Y 85.244,Z 64.500,A 180.000,B 0.000,C 180.000} C_DIS
LIN {X 88.806,Y 85.276,Z 64.500,A 180.000,B 0.000,C 180.000} C_DIS
LIN {X 88.673,Y 85.376,Z 64.500,A 180.000,B 0.000,C 180.000} C_DIS
LIN {X 88.316,Y 85.645,Z 64.500,A 180.000,B 0.000,C 180.000} C_DIS
LIN {X 88.137,Y 85.781,Z 64.500,A 180.000,B 0.000,C 180.000} C_DIS
LIN {X 88.098,Y 85.813,Z 64.500,A 180.000,B 0.000,C 180.000} C_DIS
LIN {X 87.779,Y 86.082,Z 64.500,A 180.000,B 0.000,C 180.000} C_DIS
LIN {X 87.601,Y 86.233,Z 64.500,A 180.000,B 0.000,C 180.000} C_DIS
LIN {X 87.468,Y 86.349,Z 64.500,A 180.000,B 0.000,C 180.000} C_DIS
LIN {X 87.422,Y 86.393,Z 64.500,A 180.000,B 0.000,C 180.000} C_DIS
LIN {X 87.064,Y 86.731,Z 64.500,A 180.000,B 0.000,C 180.000} C_DIS
LIN {X 86.901,Y 86.885,Z 64.500,A 180.000,B 0.000,C 180.000} C_DIS
LIN {X 86.885,Y 86.901,Z 64.500,A 180.000,B 0.000,C 180.000} C_DIS
LIN {X 86.731,Y 87.064,Z 64.500,A 180.000,B 0.000,C 180.000} C_DIS
LIN {X 86.393,Y 87.422,Z 64.500,A 180.000,B 0.000,C 180.000} C_DIS
LIN {X 86.349,Y 87.468,Z 64.500,A 180.000,B 0.000,C 180.000} C_DIS
LIN {X 86.233,Y 87.601,Z 64.500,A 180.000,B 0.000,C 180.000} C_DIS
LIN {X 85.931,Y 87.958,Z 64.500,A 180.000,B 0.000,C 180.000} C_DIS
LIN {X 85.813,Y 88.098,Z 64.500,A 180.000,B 0.000,C 180.000} C_DIS
LIN {X 85.781,Y 88.137,Z 64.500,A 180.000,B 0.000,C 180.000} C_DIS
LIN {X 85.645,Y 88.316,Z 64.500,A 180.000,B 0.000,C 180.000} C_DIS
LIN {X 85.376,Y 88.673,Z 64.500,A 180.000,B 0.000,C 180.000} C_DIS
LIN {X 85.276,Y 88.806,Z 64.500,A 180.000,B 0.000,C 180.000} C_DIS
LIN {X 85.244,Y 88.852,Z 64.500,A 180.000,B 0.000,C 180.000} C_DIS
LIN {X 85.125,Y 89.031,Z 64.500,A 180.000,B 0.000,C 180.000} C_DIS
LIN {X 84.886,Y 89.388,Z 64.500,A 180.000,B 0.000,C 180.000} C_DIS
LIN {X 84.770,Y 89.567,Z 64.500,A 180.000,B 0.000,C 180.000} C_DIS
LIN {X 84.740,Y 89.618,Z 64.500,A 180.000,B 0.000,C 180.000} C_DIS
LIN {X 84.454,Y 90.103,Z 64.500,A 180.000,B 0.000,C 180.000} C_DIS
LIN {X 84.383,Y 90.225,Z 64.500,A 180.000,B 0.000,C 180.000} C_DIS
LIN {X 84.351,Y 90.282,Z 64.500,A 180.000,B 0.000,C 180.000} C_DIS
LIN {X 84.259,Y 90.461,Z 64.500,A 180.000,B 0.000,C 180.000} C_DIS
LIN {X 84.025,Y 90.913,Z 64.500,A 180.000,B 0.000,C 180.000} C_DIS
LIN {X 83.983,Y 90.997,Z 64.500,A 180.000,B 0.000,C 180.000} C_DIS
LIN {X 83.902,Y 91.176,Z 64.500,A 180.000,B 0.000,C 180.000} C_DIS
LIN {X 83.668,Y 91.700,Z 64.500,A 180.000,B 0.000,C 180.000} C_DIS
LIN {X 83.662,Y 91.712,Z 64.500,A 180.000,B 0.000,C 180.000} C_DIS
LIN {X 83.591,Y 91.891,Z 64.500,A 180.000,B 0.000,C 180.000} C_DIS
LIN {X 83.386,Y 92.427,Z 64.500,A 180.000,B 0.000,C 180.000} C_DIS
LIN {X 83.322,Y 92.606,Z 64.500,A 180.000,B 0.000,C 180.000} C_DIS
LIN {X 83.310,Y 92.642,Z 64.500,A 180.000,B 0.000,C 180.000} C_DIS
LIN {X 83.131,Y 93.203,Z 64.500,A 180.000,B 0.000,C 180.000} C_DIS
LIN {X 83.094,Y 93.321,Z 64.500,A 180.000,B 0.000,C 180.000} C_DIS
LIN {X 83.046,Y 93.500,Z 64.500,A 180.000,B 0.000,C 180.000} C_DIS
LIN {X 82.908,Y 94.036,Z 64.500,A 180.000,B 0.000,C 180.000} C_DIS
LIN {X 82.865,Y 94.215,Z 64.500,A 180.000,B 0.000,C 180.000} C_DIS
LIN {X 82.833,Y 94.374,Z 64.500,A 180.000,B 0.000,C 180.000} C_DIS
; Link Move Starts
LIN {X 82.771,Y 94.683,Z 64.500,A 180.000,B 0.000,C 180.000} C_DIS
LIN {X 82.711,Y 94.992,Z 64.499,A 180.000,B 0.000,C 180.000} C_DIS
LIN {X 82.666,Y 95.304,Z 64.498,A 180.000,B 0.000,C 180.000} C_DIS
LIN {X 82.622,Y 95.616,Z 64.496,A 180.000,B 0.000,C 180.000} C_DIS
LIN {X 82.584,Y 95.929,Z 64.494,A 180.000,B 0.000,C 180.000} C_DIS
LIN {X 82.558,Y 96.243,Z 64.491,A 180.000,B 0.000,C 180.000} C_DIS
LIN {X 82.531,Y 96.556,Z 64.488,A 180.000,B 0.000,C 180.000} C_DIS
LIN {X 82.517,Y 96.871,Z 64.485,A 180.000,B 0.000,C 180.000} C_DIS
LIN {X 82.508,Y 97.186,Z 64.481,A 180.000,B 0.000,C 180.000} C_DIS
LIN {X 82.500,Y 97.501,Z 64.477,A 180.000,B 0.000,C 180.000} C_DIS
LIN {X 82.508,Y 97.816,Z 64.472,A 180.000,B 0.000,C 180.000} C_DIS
LIN {X 82.512,Y 97.973,Z 64.469,A 180.000,B 0.000,C 180.000} C_DIS
LIN {X 82.517,Y 98.131,Z 64.467,A 180.000,B 0.000,C 180.000} C_DIS
LIN {X 82.521,Y 98.288,Z 64.464,A 180.000,B 0.000,C 180.000} C_DIS
LIN {X 82.531,Y 98.445,Z 64.461,A 180.000,B 0.000,C 180.000} C_DIS
LIN {X 82.545,Y 98.602,Z 64.459,A 180.000,B 0.000,C 180.000} C_DIS
LIN {X 82.558,Y 98.759,Z 64.456,A 180.000,B 0.000,C 180.000} C_DIS
LIN {X 82.571,Y 98.916,Z 64.452,A 180.000,B 0.000,C 180.000} C_DIS
LIN {X 82.584,Y 99.073,Z 64.449,A 180.000,B 0.000,C 180.000} C_DIS
LIN {X 82.600,Y 99.230,Z 64.446,A 180.000,B 0.000,C 180.000} C_DIS
LIN {X 82.622,Y 99.386,Z 64.443,A 180.000,B 0.000,C 180.000} C_DIS
LIN {X 82.644,Y 99.542,Z 64.439,A 180.000,B 0.000,C 180.000} C_DIS
LIN {X 82.666,Y 99.697,Z 64.436,A 180.000,B 0.000,C 180.000} C_DIS
LIN {X 82.688,Y 99.853,Z 64.432,A 180.000,B 0.000,C 180.000} C_DIS
LIN {X 82.711,Y 100.009,Z 64.428,A 180.000,B 0.000,C 180.000} C_DIS
LIN {X 82.741,Y 100.164,Z 64.425,A 180.000,B 0.000,C 180.000} C_DIS
LIN {X 82.772,Y 100.318,Z 64.421,A 180.000,B 0.000,C 180.000} C_DIS
LIN {X 82.802,Y 100.473,Z 64.417,A 180.000,B 0.000,C 180.000} C_DIS
LIN {X 82.833,Y 100.627,Z 64.413,A 180.000,B 0.000,C 180.000} C_DIS
LIN {X 82.864,Y 100.782,Z 64.409,A 180.000,B 0.000,C 180.000} C_DIS
LIN {X 82.900,Y 100.935,Z 64.405,A 180.000,B 0.000,C 180.000} C_DIS
LIN {X 82.939,Y 101.088,Z 64.400,A 180.000,B 0.000,C 180.000} C_DIS
LIN {X 82.979,Y 101.240,Z 64.396,A 180.000,B 0.000,C 180.000} C_DIS
LIN {X 83.018,Y 101.393,Z 64.392,A 180.000,B 0.000,C 180.000} C_DIS
LIN {X 83.058,Y 101.545,Z 64.387,A 180.000,B 0.000,C 180.000} C_DIS
LIN {X 83.099,Y 101.697,Z 64.383,A 180.000,B 0.000,C 180.000} C_DIS
LIN {X 83.147,Y 101.847,Z 64.378,A 180.000,B 0.000,C 180.000} C_DIS
LIN {X 83.195,Y 101.997,Z 64.373,A 180.000,B 0.000,C 180.000} C_DIS
LIN {X 83.243,Y 102.147,Z 64.369,A 180.000,B 0.000,C 180.000} C_DIS
LIN {X 83.291,Y 102.297,Z 64.364,A 180.000,B 0.000,C 180.000} C_DIS
LIN {X 83.339,Y 102.447,Z 64.359,A 180.000,B 0.000,C 180.000} C_DIS
LIN {X 83.394,Y 102.595,Z 64.354,A 180.000,B 0.000,C 180.000} C_DIS
LIN {X 83.422,Y 102.668,Z 64.351,A 180.000,B 0.000,C 180.000} C_DIS
LIN {X 83.450,Y 102.742,Z 64.349,A 180.000,B 0.000,C 180.000} C_DIS
LIN {X 83.479,Y 102.815,Z 64.346,A 180.000,B 0.000,C 180.000} C_DIS
LIN {X 83.507,Y 102.889,Z 64.344,A 180.000,B 0.000,C 180.000} C_DIS
LIN {X 83.535,Y 102.962,Z 64.341,A 180.000,B 0.000,C 180.000} C_DIS
LIN {X 83.563,Y 103.036,Z 64.339,A 180.000,B 0.000,C 180.000} C_DIS
LIN {X 83.591,Y 103.110,Z 64.336,A 180.000,B 0.000,C 180.000} C_DIS
LIN {X 83.619,Y 103.183,Z 64.333,A 180.000,B 0.000,C 180.000} C_DIS
LIN {X 83.648,Y 103.256,Z 64.331,A 180.000,B 0.000,C 180.000} C_DIS
LIN {X 83.680,Y 103.328,Z 64.328,A 180.000,B 0.000,C 180.000} C_DIS
LIN {X 83.744,Y 103.472,Z 64.323,A 180.000,B 0.000,C 180.000} C_DIS
LIN {X 83.809,Y 103.616,Z 64.317,A 180.000,B 0.000,C 180.000} C_DIS
LIN {X 83.873,Y 103.760,Z 64.312,A 180.000,B 0.000,C 180.000} C_DIS
LIN {X 83.937,Y 103.903,Z 64.307,A 180.000,B 0.000,C 180.000} C_DIS
LIN {X 83.970,Y 103.975,Z 64.304,A 180.000,B 0.000,C 180.000} C_DIS
LIN {X 84.004,Y 104.046,Z 64.301,A 180.000,B 0.000,C 180.000} C_DIS
LIN {X 84.040,Y 104.116,Z 64.298,A 180.000,B 0.000,C 180.000} C_DIS
LIN {X 84.076,Y 104.186,Z 64.296,A 180.000,B 0.000,C 180.000} C_DIS
LIN {X 84.149,Y 104.326,Z 64.290,A 180.000,B 0.000,C 180.000} C_DIS
LIN {X 84.257,Y 104.536,Z 64.282,A 180.000,B 0.000,C 180.000} C_DIS
LIN {X 84.329,Y 104.676,Z 64.276,A 180.000,B 0.000,C 180.000} C_DIS
LIN {X 84.366,Y 104.746,Z 64.274,A 180.000,B 0.000,C 180.000} C_DIS
LIN {X 84.405,Y 104.814,Z 64.271,A 180.000,B 0.000,C 180.000} C_DIS
LIN {X 84.485,Y 104.950,Z 64.265,A 180.000,B 0.000,C 180.000} C_DIS
LIN {X 84.525,Y 105.018,Z 64.263,A 180.000,B 0.000,C 180.000} C_DIS
LIN {X 84.605,Y 105.153,Z 64.257,A 180.000,B 0.000,C 180.000} C_DIS
LIN {X 84.725,Y 105.357,Z 64.249,A 180.000,B 0.000,C 180.000} C_DIS
LIN {X 84.765,Y 105.424,Z 64.246,A 180.000,B 0.000,C 180.000} C_DIS
LIN {X 84.806,Y 105.492,Z 64.243,A 180.000,B 0.000,C 180.000} C_DIS
LIN {X 84.849,Y 105.557,Z 64.241,A 180.000,B 0.000,C 180.000} C_DIS
LIN {X 84.937,Y 105.688,Z 64.235,A 180.000,B 0.000,C 180.000} C_DIS
LIN {X 85.068,Y 105.885,Z 64.227,A 180.000,B 0.000,C 180.000} C_DIS
LIN {X 85.156,Y 106.016,Z 64.221,A 180.000,B 0.000,C 180.000} C_DIS
LIN {X 85.199,Y 106.081,Z 64.219,A 180.000,B 0.000,C 180.000} C_DIS
LIN {X 85.243,Y 106.147,Z 64.216,A 180.000,B 0.000,C 180.000} C_DIS
LIN {X 85.289,Y 106.211,Z 64.213,A 180.000,B 0.000,C 180.000} C_DIS
LIN {X 85.336,Y 106.274,Z 64.210,A 180.000,B 0.000,C 180.000} C_DIS
LIN {X 85.383,Y 106.337,Z 64.208,A 180.000,B 0.000,C 180.000} C_DIS
LIN {X 85.478,Y 106.463,Z 64.202,A 180.000,B 0.000,C 180.000} C_DIS
LIN {X 85.715,Y 106.777,Z 64.188,A 180.000,B 0.000,C 180.000} C_DIS
LIN {X 85.763,Y 106.840,Z 64.186,A 180.000,B 0.000,C 180.000} C_DIS
LIN {X 85.812,Y 106.901,Z 64.183,A 180.000,B 0.000,C 180.000} C_DIS
LIN {X 85.914,Y 107.021,Z 64.177,A 180.000,B 0.000,C 180.000} C_DIS
LIN {X 85.965,Y 107.082,Z 64.175,A 180.000,B 0.000,C 180.000} C_DIS
LIN {X 86.066,Y 107.202,Z 64.169,A 180.000,B 0.000,C 180.000} C_DIS
LIN {X 86.270,Y 107.443,Z 64.158,A 180.000,B 0.000,C 180.000} C_DIS
LIN {X 86.321,Y 107.502,Z 64.155,A 180.000,B 0.000,C 180.000} C_DIS
LIN {X 86.375,Y 107.560,Z 64.153,A 180.000,B 0.000,C 180.000} C_DIS
LIN {X 86.537,Y 107.731,Z 64.144,A 180.000,B 0.000,C 180.000} C_DIS
LIN {X 86.645,Y 107.846,Z 64.139,A 180.000,B 0.000,C 180.000} C_DIS
LIN {X 86.808,Y 108.017,Z 64.131,A 180.000,B 0.000,C 180.000} C_DIS
LIN {X 86.862,Y 108.075,Z 64.128,A 180.000,B 0.000,C 180.000} C_DIS
LIN {X 86.917,Y 108.130,Z 64.125,A 180.000,B 0.000,C 180.000} C_DIS
LIN {X 86.975,Y 108.185,Z 64.122,A 180.000,B 0.000,C 180.000} C_DIS
LIN {X 87.089,Y 108.293,Z 64.117,A 180.000,B 0.000,C 180.000} C_DIS
LIN {X 87.432,Y 108.617,Z 64.100,A 180.000,B 0.000,C 180.000} C_DIS
LIN {X 87.490,Y 108.671,Z 64.098,A 180.000,B 0.000,C 180.000} C_DIS
LIN {X 87.549,Y 108.723,Z 64.095,A 180.000,B 0.000,C 180.000} C_DIS
LIN {X 87.609,Y 108.774,Z 64.092,A 180.000,B 0.000,C 180.000} C_DIS
LIN {X 88.090,Y 109.180,Z 64.070,A 180.000,B 0.000,C 180.000} C_DIS
LIN {X 88.151,Y 109.230,Z 64.067,A 180.000,B 0.000,C 180.000} C_DIS
LIN {X 88.214,Y 109.278,Z 64.065,A 180.000,B 0.000,C 180.000} C_DIS
LIN {X 88.591,Y 109.563,Z 64.048,A 180.000,B 0.000,C 180.000} C_DIS
LIN {X 88.717,Y 109.657,Z 64.043,A 180.000,B 0.000,C 180.000} C_DIS
LIN {X 88.780,Y 109.705,Z 64.040,A 180.000,B 0.000,C 180.000} C_DIS
LIN {X 88.844,Y 109.750,Z 64.037,A 180.000,B 0.000,C 180.000} C_DIS
LIN {X 88.909,Y 109.794,Z 64.034,A 180.000,B 0.000,C 180.000} C_DIS
LIN {X 89.433,Y 110.144,Z 64.012,A 180.000,B 0.000,C 180.000} C_DIS
LIN {X 89.499,Y 110.188,Z 64.010,A 180.000,B 0.000,C 180.000} C_DIS
LIN {X 89.566,Y 110.229,Z 64.007,A 180.000,B 0.000,C 180.000} C_DIS
LIN {X 89.634,Y 110.269,Z 64.004,A 180.000,B 0.000,C 180.000} C_DIS
LIN {X 90.176,Y 110.589,Z 63.982,A 180.000,B 0.000,C 180.000} C_DIS
LIN {X 90.245,Y 110.629,Z 63.979,A 180.000,B 0.000,C 180.000} C_DIS
LIN {X 90.314,Y 110.666,Z 63.977,A 180.000,B 0.000,C 180.000} C_DIS
LIN {X 90.874,Y 110.955,Z 63.955,A 180.000,B 0.000,C 180.000} C_DIS
LIN {X 90.944,Y 110.991,Z 63.952,A 180.000,B 0.000,C 180.000} C_DIS
LIN {X 91.015,Y 111.025,Z 63.949,A 180.000,B 0.000,C 180.000} C_DIS
LIN {X 91.086,Y 111.058,Z 63.946,A 180.000,B 0.000,C 180.000} C_DIS
LIN {X 91.446,Y 111.219,Z 63.933,A 180.000,B 0.000,C 180.000} C_DIS
LIN {X 91.662,Y 111.315,Z 63.924,A 180.000,B 0.000,C 180.000} C_DIS
LIN {X 91.734,Y 111.347,Z 63.922,A 180.000,B 0.000,C 180.000} C_DIS
LIN {X 91.806,Y 111.377,Z 63.919,A 180.000,B 0.000,C 180.000} C_DIS
LIN {X 91.880,Y 111.405,Z 63.916,A 180.000,B 0.000,C 180.000} C_DIS
LIN {X 92.469,Y 111.630,Z 63.894,A 180.000,B 0.000,C 180.000} C_DIS
LIN {X 92.542,Y 111.657,Z 63.891,A 180.000,B 0.000,C 180.000} C_DIS
LIN {X 92.617,Y 111.682,Z 63.889,A 180.000,B 0.000,C 180.000} C_DIS
LIN {X 92.842,Y 111.754,Z 63.880,A 180.000,B 0.000,C 180.000} C_DIS
LIN {X 92.992,Y 111.802,Z 63.875,A 180.000,B 0.000,C 180.000} C_DIS
LIN {X 93.217,Y 111.873,Z 63.867,A 180.000,B 0.000,C 180.000} C_DIS
LIN {X 93.292,Y 111.897,Z 63.864,A 180.000,B 0.000,C 180.000} C_DIS
LIN {X 93.368,Y 111.920,Z 63.861,A 180.000,B 0.000,C 180.000} C_DIS
LIN {X 93.444,Y 111.940,Z 63.858,A 180.000,B 0.000,C 180.000} C_DIS
LIN {X 93.597,Y 111.979,Z 63.853,A 180.000,B 0.000,C 180.000} C_DIS
LIN {X 94.054,Y 112.097,Z 63.836,A 180.000,B 0.000,C 180.000} C_DIS
LIN {X 94.130,Y 112.116,Z 63.834,A 180.000,B 0.000,C 180.000} C_DIS
LIN {X 94.207,Y 112.134,Z 63.831,A 180.000,B 0.000,C 180.000} C_DIS
LIN {X 94.284,Y 112.149,Z 63.828,A 180.000,B 0.000,C 180.000} C_DIS
LIN {X 94.748,Y 112.241,Z 63.812,A 180.000,B 0.000,C 180.000} C_DIS
LIN {X 94.902,Y 112.272,Z 63.806,A 180.000,B 0.000,C 180.000} C_DIS
LIN {X 94.980,Y 112.287,Z 63.803,A 180.000,B 0.000,C 180.000} C_DIS
LIN {X 95.058,Y 112.299,Z 63.801,A 180.000,B 0.000,C 180.000} C_DIS
LIN {X 95.214,Y 112.321,Z 63.795,A 180.000,B 0.000,C 180.000} C_DIS
LIN {X 95.681,Y 112.387,Z 63.779,A 180.000,B 0.000,C 180.000} C_DIS
LIN {X 95.759,Y 112.398,Z 63.776,A 180.000,B 0.000,C 180.000} C_DIS
LIN {X 95.838,Y 112.408,Z 63.773,A 180.000,B 0.000,C 180.000} C_DIS
LIN {X 95.916,Y 112.415,Z 63.770,A 180.000,B 0.000,C 180.000} C_DIS
LIN {X 95.994,Y 112.421,Z 63.768,A 180.000,B 0.000,C 180.000} C_DIS
LIN {X 96.151,Y 112.435,Z 63.762,A 180.000,B 0.000,C 180.000} C_DIS
LIN {X 96.387,Y 112.454,Z 63.754,A 180.000,B 0.000,C 180.000} C_DIS
LIN {X 96.544,Y 112.468,Z 63.748,A 180.000,B 0.000,C 180.000} C_DIS
LIN {X 96.622,Y 112.474,Z 63.746,A 180.000,B 0.000,C 180.000} C_DIS
LIN {X 96.701,Y 112.478,Z 63.743,A 180.000,B 0.000,C 180.000} C_DIS
LIN {X 96.780,Y 112.481,Z 63.740,A 180.000,B 0.000,C 180.000} C_DIS
LIN {X 97.016,Y 112.487,Z 63.732,A 180.000,B 0.000,C 180.000} C_DIS
LIN {X 97.173,Y 112.492,Z 63.726,A 180.000,B 0.000,C 180.000} C_DIS
LIN {X 97.252,Y 112.494,Z 63.724,A 180.000,B 0.000,C 180.000} C_DIS
LIN {X 97.409,Y 112.498,Z 63.718,A 180.000,B 0.000,C 180.000} C_DIS
LIN {X 97.488,Y 112.500,Z 63.715,A 180.000,B 0.000,C 180.000} C_DIS
LIN {X 97.567,Y 112.499,Z 63.713,A 180.000,B 0.000,C 180.000} C_DIS
LIN {X 97.724,Y 112.495,Z 63.707,A 180.000,B 0.000,C 180.000} C_DIS
LIN {X 97.960,Y 112.488,Z 63.699,A 180.000,B 0.000,C 180.000} C_DIS
LIN {X 98.118,Y 112.484,Z 63.693,A 180.000,B 0.000,C 180.000} C_DIS
LIN {X 98.275,Y 112.479,Z 63.688,A 180.000,B 0.000,C 180.000} C_DIS
LIN {X 98.354,Y 112.476,Z 63.685,A 180.000,B 0.000,C 180.000} C_DIS
LIN {X 98.433,Y 112.470,Z 63.682,A 180.000,B 0.000,C 180.000} C_DIS
LIN {X 98.589,Y 112.456,Z 63.677,A 180.000,B 0.000,C 180.000} C_DIS
LIN {X 98.746,Y 112.443,Z 63.672,A 180.000,B 0.000,C 180.000} C_DIS
LIN {X 98.903,Y 112.430,Z 63.666,A 180.000,B 0.000,C 180.000} C_DIS
LIN {X 98.982,Y 112.423,Z 63.664,A 180.000,B 0.000,C 180.000} C_DIS
LIN {X 99.060,Y 112.417,Z 63.661,A 180.000,B 0.000,C 180.000} C_DIS
LIN {X 99.139,Y 112.410,Z 63.659,A 180.000,B 0.000,C 180.000} C_DIS
LIN {X 99.217,Y 112.401,Z 63.656,A 180.000,B 0.000,C 180.000} C_DIS
LIN {X 99.295,Y 112.390,Z 63.654,A 180.000,B 0.000,C 180.000} C_DIS
LIN {X 99.373,Y 112.379,Z 63.651,A 180.000,B 0.000,C 180.000} C_DIS
LIN {X 99.451,Y 112.368,Z 63.649,A 180.000,B 0.000,C 180.000} C_DIS
LIN {X 99.607,Y 112.346,Z 63.644,A 180.000,B 0.000,C 180.000} C_DIS
LIN {X 99.763,Y 112.324,Z 63.639,A 180.000,B 0.000,C 180.000} C_DIS
LIN {X 99.919,Y 112.302,Z 63.634,A 180.000,B 0.000,C 180.000} C_DIS
LIN {X 100.074,Y 112.277,Z 63.629,A 180.000,B 0.000,C 180.000} C_DIS
LIN {X 100.229,Y 112.246,Z 63.624,A 180.000,B 0.000,C 180.000} C_DIS
LIN {X 100.383,Y 112.215,Z 63.620,A 180.000,B 0.000,C 180.000} C_DIS
LIN {X 100.538,Y 112.185,Z 63.615,A 180.000,B 0.000,C 180.000} C_DIS
LIN {X 100.692,Y 112.154,Z 63.610,A 180.000,B 0.000,C 180.000} C_DIS
LIN {X 100.846,Y 112.122,Z 63.606,A 180.000,B 0.000,C 180.000} C_DIS
LIN {X 100.999,Y 112.083,Z 63.602,A 180.000,B 0.000,C 180.000} C_DIS
LIN {X 101.152,Y 112.044,Z 63.597,A 180.000,B 0.000,C 180.000} C_DIS
LIN {X 101.304,Y 112.005,Z 63.593,A 180.000,B 0.000,C 180.000} C_DIS
LIN {X 101.457,Y 111.965,Z 63.589,A 180.000,B 0.000,C 180.000} C_DIS
LIN {X 101.609,Y 111.926,Z 63.585,A 180.000,B 0.000,C 180.000} C_DIS
LIN {X 101.760,Y 111.881,Z 63.581,A 180.000,B 0.000,C 180.000} C_DIS
LIN {X 101.910,Y 111.833,Z 63.577,A 180.000,B 0.000,C 180.000} C_DIS
LIN {X 102.060,Y 111.785,Z 63.573,A 180.000,B 0.000,C 180.000} C_DIS
LIN {X 102.210,Y 111.737,Z 63.570,A 180.000,B 0.000,C 180.000} C_DIS
LIN {X 102.360,Y 111.689,Z 63.566,A 180.000,B 0.000,C 180.000} C_DIS
LIN {X 102.509,Y 111.638,Z 63.562,A 180.000,B 0.000,C 180.000} C_DIS
LIN {X 102.656,Y 111.582,Z 63.559,A 180.000,B 0.000,C 180.000} C_DIS
LIN {X 102.803,Y 111.526,Z 63.556,A 180.000,B 0.000,C 180.000} C_DIS
LIN {X 102.951,Y 111.470,Z 63.552,A 180.000,B 0.000,C 180.000} C_DIS
LIN {X 103.098,Y 111.414,Z 63.549,A 180.000,B 0.000,C 180.000} C_DIS
LIN {X 103.245,Y 111.356,Z 63.546,A 180.000,B 0.000,C 180.000} C_DIS
LIN {X 103.389,Y 111.293,Z 63.543,A 180.000,B 0.000,C 180.000} C_DIS
LIN {X 103.532,Y 111.229,Z 63.540,A 180.000,B 0.000,C 180.000} C_DIS
LIN {X 103.676,Y 111.164,Z 63.537,A 180.000,B 0.000,C 180.000} C_DIS
LIN {X 103.820,Y 111.100,Z 63.534,A 180.000,B 0.000,C 180.000} C_DIS
LIN {X 103.964,Y 111.035,Z 63.532,A 180.000,B 0.000,C 180.000} C_DIS
LIN {X 104.105,Y 110.966,Z 63.529,A 180.000,B 0.000,C 180.000} C_DIS
LIN {X 104.245,Y 110.893,Z 63.527,A 180.000,B 0.000,C 180.000} C_DIS
LIN {X 104.525,Y 110.749,Z 63.522,A 180.000,B 0.000,C 180.000} C_DIS
LIN {X 104.803,Y 110.602,Z 63.518,A 180.000,B 0.000,C 180.000} C_DIS
LIN {X 105.074,Y 110.442,Z 63.514,A 180.000,B 0.000,C 180.000} C_DIS
LIN {X 105.346,Y 110.282,Z 63.511,A 180.000,B 0.000,C 180.000} C_DIS
LIN {X 105.612,Y 110.114,Z 63.508,A 180.000,B 0.000,C 180.000} C_DIS
LIN {X 105.874,Y 109.939,Z 63.505,A 180.000,B 0.000,C 180.000} C_DIS
LIN {X 106.136,Y 109.764,Z 63.503,A 180.000,B 0.000,C 180.000} C_DIS
LIN {X 106.390,Y 109.577,Z 63.502,A 180.000,B 0.000,C 180.000} C_DIS
LIN {X 106.641,Y 109.388,Z 63.501,A 180.000,B 0.000,C 180.000} C_DIS
LIN {X 106.891,Y 109.196,Z 63.500,A 180.000,B 0.000,C 180.000} C_DIS
LIN {X 107.068,Y 109.046,Z 63.500,A 180.000,B 0.000,C 180.000} C_DIS
; Cutting Move Starts
LIN {X 107.444,Y 108.729,Z 63.500,A 180.000,B 0.000,C 180.000} C_DIS
LIN {X 107.483,Y 108.695,Z 63.500,A 180.000,B 0.000,C 180.000} C_DIS
LIN {X 107.623,Y 108.565,Z 63.500,A 180.000,B 0.000,C 180.000} C_DIS
LIN {X 108.053,Y 108.159,Z 63.500,A 180.000,B 0.000,C 180.000} C_DIS
LIN {X 108.159,Y 108.053,Z 63.500,A 180.000,B 0.000,C 180.000} C_DIS
LIN {X 108.565,Y 107.623,Z 63.500,A 180.000,B 0.000,C 180.000} C_DIS
LIN {X 108.695,Y 107.483,Z 63.500,A 180.000,B 0.000,C 180.000} C_DIS
LIN {X 108.729,Y 107.444,Z 63.500,A 180.000,B 0.000,C 180.000} C_DIS
LIN {X 109.182,Y 106.908,Z 63.500,A 180.000,B 0.000,C 180.000} C_DIS
LIN {X 109.232,Y 106.847,Z 63.500,A 180.000,B 0.000,C 180.000} C_DIS
LIN {X 109.322,Y 106.729,Z 63.500,A 180.000,B 0.000,C 180.000} C_DIS
LIN {X 109.591,Y 106.371,Z 63.500,A 180.000,B 0.000,C 180.000} C_DIS
LIN {X 109.724,Y 106.193,Z 63.500,A 180.000,B 0.000,C 180.000} C_DIS
LIN {X 109.768,Y 106.130,Z 63.500,A 180.000,B 0.000,C 180.000} C_DIS
LIN {X 109.846,Y 106.014,Z 63.500,A 180.000,B 0.000,C 180.000} C_DIS
LIN {X 110.126,Y 105.595,Z 63.500,A 180.000,B 0.000,C 180.000} C_DIS
LIN {X 110.203,Y 105.477,Z 63.500,A 180.000,B 0.000,C 180.000} C_DIS
LIN {X 110.304,Y 105.307,Z 63.500,A 180.000,B 0.000,C 180.000} C_DIS
LIN {X 110.520,Y 104.941,Z 63.500,A 180.000,B 0.000,C 180.000} C_DIS
LIN {X 110.625,Y 104.762,Z 63.500,A 180.000,B 0.000,C 180.000} C_DIS
LIN {X 110.662,Y 104.693,Z 63.500,A 180.000,B 0.000,C 180.000} C_DIS
LIN {X 110.903,Y 104.226,Z 63.500,A 180.000,B 0.000,C 180.000} C_DIS
LIN {X 110.995,Y 104.047,Z 63.500,A 180.000,B 0.000,C 180.000} C_DIS
LIN {X 111.019,Y 103.998,Z 63.500,A 180.000,B 0.000,C 180.000} C_DIS
LIN {X 111.078,Y 103.869,Z 63.500,A 180.000,B 0.000,C 180.000} C_DIS
LIN {X 111.318,Y 103.332,Z 63.500,A 180.000,B 0.000,C 180.000} C_DIS
LIN {X 111.377,Y 103.194,Z 63.500,A 180.000,B 0.000,C 180.000} C_DIS
LIN {X 111.392,Y 103.153,Z 63.500,A 180.000,B 0.000,C 180.000} C_DIS
LIN {X 111.597,Y 102.617,Z 63.500,A 180.000,B 0.000,C 180.000} C_DIS
LIN {X 111.664,Y 102.438,Z 63.500,A 180.000,B 0.000,C 180.000} C_DIS
LIN {X 111.721,Y 102.260,Z 63.500,A 180.000,B 0.000,C 180.000} C_DIS
LIN {X 111.892,Y 101.723,Z 63.500,A 180.000,B 0.000,C 180.000} C_DIS
LIN {X 111.913,Y 101.654,Z 63.500,A 180.000,B 0.000,C 180.000} C_DIS
LIN {X 111.943,Y 101.545,Z 63.500,A 180.000,B 0.000,C 180.000} C_DIS
LIN {X 112.092,Y 100.966,Z 63.500,A 180.000,B 0.000,C 180.000} C_DIS
LIN {X 112.126,Y 100.829,Z 63.500,A 180.000,B 0.000,C 180.000} C_DIS
LIN {X 112.162,Y 100.651,Z 63.500,A 180.000,B 0.000,C 180.000} C_DIS
LIN {X 112.271,Y 100.105,Z 63.500,A 180.000,B 0.000,C 180.000} C_DIS
LIN {X 112.300,Y 99.936,Z 63.500,A 180.000,B 0.000,C 180.000} C_DIS
LIN {X 112.376,Y 99.399,Z 63.500,A 180.000,B 0.000,C 180.000} C_DIS
LIN {X 112.401,Y 99.221,Z 63.500,A 180.000,B 0.000,C 180.000} C_DIS
LIN {X 112.418,Y 99.042,Z 63.500,A 180.000,B 0.000,C 180.000} C_DIS
LIN {X 112.464,Y 98.505,Z 63.500,A 180.000,B 0.000,C 180.000} C_DIS
LIN {X 112.477,Y 98.327,Z 63.500,A 180.000,B 0.000,C 180.000} C_DIS
LIN {X 112.483,Y 98.148,Z 63.500,A 180.000,B 0.000,C 180.000} C_DIS
LIN {X 112.498,Y 97.612,Z 63.500,A 180.000,B 0.000,C 180.000} C_DIS
LIN {X 112.499,Y 97.433,Z 63.500,A 180.000,B 0.000,C 180.000} C_DIS
LIN {X 112.484,Y 96.897,Z 63.500,A 180.000,B 0.000,C 180.000} C_DIS
LIN {X 112.479,Y 96.718,Z 63.500,A 180.000,B 0.000,C 180.000} C_DIS
LIN {X 112.467,Y 96.539,Z 63.500,A 180.000,B 0.000,C 180.000} C_DIS
LIN {X 112.422,Y 96.003,Z 63.500,A 180.000,B 0.000,C 180.000} C_DIS
LIN {X 112.406,Y 95.824,Z 63.500,A 180.000,B 0.000,C 180.000} C_DIS
LIN {X 112.382,Y 95.645,Z 63.500,A 180.000,B 0.000,C 180.000} C_DIS
LIN {X 112.306,Y 95.109,Z 63.500,A 180.000,B 0.000,C 180.000} C_DIS
LIN {X 112.278,Y 94.930,Z 63.500,A 180.000,B 0.000,C 180.000} C_DIS
LIN {X 112.271,Y 94.895,Z 63.500,A 180.000,B 0.000,C 180.000} C_DIS
LIN {X 112.171,Y 94.394,Z 63.500,A 180.000,B 0.000,C 180.000} C_DIS
LIN {X 112.135,Y 94.215,Z 63.500,A 180.000,B 0.000,C 180.000} C_DIS
LIN {X 112.092,Y 94.036,Z 63.500,A 180.000,B 0.000,C 180.000} C_DIS
LIN {X 111.954,Y 93.500,Z 63.500,A 180.000,B 0.000,C 180.000} C_DIS
LIN {X 111.913,Y 93.346,Z 63.500,A 180.000,B 0.000,C 180.000} C_DIS
LIN {X 111.906,Y 93.321,Z 63.500,A 180.000,B 0.000,C 180.000} C_DIS
LIN {X 111.849,Y 93.142,Z 63.500,A 180.000,B 0.000,C 180.000} C_DIS
LIN {X 111.734,Y 92.782,Z 63.500,A 180.000,B 0.000,C 180.000} C_DIS
LIN {X 111.678,Y 92.606,Z 63.500,A 180.000,B 0.000,C 180.000} C_DIS
LIN {X 111.614,Y 92.427,Z 63.500,A 180.000,B 0.000,C 180.000} C_DIS
LIN {X 111.409,Y 91.891,Z 63.500,A 180.000,B 0.000,C 180.000} C_DIS
LIN {X 111.377,Y 91.806,Z 63.500,A 180.000,B 0.000,C 180.000} C_DIS
LIN {X 111.338,Y 91.712,Z 63.500,A 180.000,B 0.000,C 180.000} C_DIS
LIN {X 111.258,Y 91.533,Z 63.500,A 180.000,B 0.000,C 180.000} C_DIS
LIN {X 111.098,Y 91.176,Z 63.500,A 180.000,B 0.000,C 180.000} C_DIS
LIN {X 111.019,Y 91.002,Z 63.500,A 180.000,B 0.000,C 180.000} C_DIS
LIN {X 111.017,Y 90.997,Z 63.500,A 180.000,B 0.000,C 180.000} C_DIS
LIN {X 110.926,Y 90.818,Z 63.500,A 180.000,B 0.000,C 180.000} C_DIS
LIN {X 110.662,Y 90.307,Z 63.500,A 180.000,B 0.000,C 180.000} C_DIS
LIN {X 110.649,Y 90.282,Z 63.500,A 180.000,B 0.000,C 180.000} C_DIS
LIN {X 110.546,Y 90.103,Z 63.500,A 180.000,B 0.000,C 180.000} C_DIS
LIN {X 110.304,Y 89.693,Z 63.500,A 180.000,B 0.000,C 180.000} C_DIS
LIN {X 110.230,Y 89.567,Z 63.500,A 180.000,B 0.000,C 180.000} C_DIS
LIN {X 110.126,Y 89.405,Z 63.500,A 180.000,B 0.000,C 180.000} C_DIS
LIN {X 109.875,Y 89.031,Z 63.500,A 180.000,B 0.000,C 180.000} C_DIS
LIN {X 109.768,Y 88.870,Z 63.500,A 180.000,B 0.000,C 180.000} C_DIS
LIN {X 109.756,Y 88.852,Z 63.500,A 180.000,B 0.000,C 180.000} C_DIS
LIN {X 109.624,Y 88.673,Z 63.500,A 180.000,B 0.000,C 180.000} C_DIS
LIN {X 109.355,Y 88.316,Z 63.500,A 180.000,B 0.000,C 180.000} C_DIS
LIN {X 109.232,Y 88.153,Z 63.500,A 180.000,B 0.000,C 180.000} C_DIS
LIN {X 109.219,Y 88.137,Z 63.500,A 180.000,B 0.000,C 180.000} C_DIS
LIN {X 109.069,Y 87.958,Z 63.500,A 180.000,B 0.000,C 180.000} C_DIS
LIN {X 108.767,Y 87.601,Z 63.500,A 180.000,B 0.000,C 180.000} C_DIS
LIN {X 108.695,Y 87.517,Z 63.500,A 180.000,B 0.000,C 180.000} C_DIS
LIN {X 108.607,Y 87.422,Z 63.500,A 180.000,B 0.000,C 180.000} C_DIS
LIN {X 108.159,Y 86.947,Z 63.500,A 180.000,B 0.000,C 180.000} C_DIS
LIN {X 108.099,Y 86.885,Z 63.500,A 180.000,B 0.000,C 180.000} C_DIS
LIN {X 107.980,Y 86.773,Z 63.500,A 180.000,B 0.000,C 180.000} C_DIS
LIN {X 107.623,Y 86.435,Z 63.500,A 180.000,B 0.000,C 180.000} C_DIS
LIN {X 107.532,Y 86.349,Z 63.500,A 180.000,B 0.000,C 180.000} C_DIS
LIN {X 107.444,Y 86.271,Z 63.500,A 180.000,B 0.000,C 180.000} C_DIS
LIN {X 106.908,Y 85.818,Z 63.500,A 180.000,B 0.000,C 180.000} C_DIS
LIN {X 106.902,Y 85.813,Z 63.500,A 180.000,B 0.000,C 180.000} C_DIS
LIN {X 106.729,Y 85.678,Z 63.500,A 180.000,B 0.000,C 180.000} C_DIS
LIN {X 106.371,Y 85.409,Z 63.500,A 180.000,B 0.000,C 180.000} C_DIS
LIN {X 106.194,Y 85.276,Z 63.500,A 180.000,B 0.000,C 180.000} C_DIS
LIN {X 106.193,Y 85.276,Z 63.500,A 180.000,B 0.000,C 180.000} C_DIS
LIN {X 106.014,Y 85.154,Z 63.500,A 180.000,B 0.000,C 180.000} C_DIS
LIN {X 105.656,Y 84.915,Z 63.500,A 180.000,B 0.000,C 180.000} C_DIS
LIN {X 105.477,Y 84.797,Z 63.500,A 180.000,B 0.000,C 180.000} C_DIS
LIN {X 105.382,Y 84.740,Z 63.500,A 180.000,B 0.000,C 180.000} C_DIS
LIN {X 104.941,Y 84.480,Z 63.500,A 180.000,B 0.000,C 180.000} C_DIS
LIN {X 104.775,Y 84.383,Z 63.500,A 180.000,B 0.000,C 180.000} C_DIS
LIN {X 104.762,Y 84.375,Z 63.500,A 180.000,B 0.000,C 180.000} C_DIS
LIN {X 104.584,Y 84.282,Z 63.500,A 180.000,B 0.000,C 180.000} C_DIS
LIN {X 104.087,Y 84.025,Z 63.500,A 180.000,B 0.000,C 180.000} C_DIS
LIN {X 104.047,Y 84.005,Z 63.500,A 180.000,B 0.000,C 180.000} C_DIS
LIN {X 103.869,Y 83.922,Z 63.500,A 180.000,B 0.000,C 180.000} C_DIS
LIN {X 103.300,Y 83.668,Z 63.500,A 180.000,B 0.000,C 180.000} C_DIS
LIN {X 103.153,Y 83.608,Z 63.500,A 180.000,B 0.000,C 180.000} C_DIS
LIN {X 102.617,Y 83.403,Z 63.500,A 180.000,B 0.000,C 180.000} C_DIS
LIN {X 102.438,Y 83.336,Z 63.500,A 180.000,B 0.000,C 180.000} C_DIS
LIN {X 102.358,Y 83.310,Z 63.500,A 180.000,B 0.000,C 180.000} C_DIS
LIN {X 101.723,Y 83.108,Z 63.500,A 180.000,B 0.000,C 180.000} C_DIS
LIN {X 101.545,Y 83.057,Z 63.500,A 180.000,B 0.000,C 180.000} C_DIS
LIN {X 101.008,Y 82.919,Z 63.500,A 180.000,B 0.000,C 180.000} C_DIS
LIN {X 100.829,Y 82.874,Z 63.500,A 180.000,B 0.000,C 180.000} C_DIS
LIN {X 100.651,Y 82.838,Z 63.500,A 180.000,B 0.000,C 180.000} C_DIS
LIN {X 100.114,Y 82.731,Z 63.500,A 180.000,B 0.000,C 180.000} C_DIS
LIN {X 99.936,Y 82.700,Z 63.500,A 180.000,B 0.000,C 180.000} C_DIS
LIN {X 99.399,Y 82.624,Z 63.500,A 180.000,B 0.000,C 180.000} C_DIS
LIN {X 99.221,Y 82.599,Z 63.500,A 180.000,B 0.000,C 180.000} C_DIS
LIN {X 99.185,Y 82.595,Z 63.500,A 180.000,B 0.000,C 180.000} C_DIS
LIN {X 99.042,Y 82.582,Z 63.500,A 180.000,B 0.000,C 180.000} C_DIS
LIN {X 98.505,Y 82.536,Z 63.500,A 180.000,B 0.000,C 180.000} C_DIS
LIN {X 98.327,Y 82.523,Z 63.500,A 180.000,B 0.000,C 180.000} C_DIS
LIN {X 98.148,Y 82.517,Z 63.500,A 180.000,B 0.000,C 180.000} C_DIS
LIN {X 97.612,Y 82.502,Z 63.500,A 180.000,B 0.000,C 180.000} C_DIS
LIN {X 97.433,Y 82.501,Z 63.500,A 180.000,B 0.000,C 180.000} C_DIS
LIN {X 96.897,Y 82.516,Z 63.500,A 180.000,B 0.000,C 180.000} C_DIS
LIN {X 96.718,Y 82.521,Z 63.500,A 180.000,B 0.000,C 180.000} C_DIS
LIN {X 96.539,Y 82.533,Z 63.500,A 180.000,B 0.000,C 180.000} C_DIS
LIN {X 96.003,Y 82.578,Z 63.500,A 180.000,B 0.000,C 180.000} C_DIS
LIN {X 95.824,Y 82.594,Z 63.500,A 180.000,B 0.000,C 180.000} C_DIS
LIN {X 95.815,Y 82.595,Z 63.500,A 180.000,B 0.000,C 180.000} C_DIS
LIN {X 95.645,Y 82.618,Z 63.500,A 180.000,B 0.000,C 180.000} C_DIS
LIN {X 95.109,Y 82.694,Z 63.500,A 180.000,B 0.000,C 180.000} C_DIS
LIN {X 94.930,Y 82.722,Z 63.500,A 180.000,B 0.000,C 180.000} C_DIS
LIN {X 94.751,Y 82.758,Z 63.500,A 180.000,B 0.000,C 180.000} C_DIS
LIN {X 94.394,Y 82.829,Z 63.500,A 180.000,B 0.000,C 180.000} C_DIS
LIN {X 94.215,Y 82.865,Z 63.500,A 180.000,B 0.000,C 180.000} C_DIS
LIN {X 94.036,Y 82.908,Z 63.500,A 180.000,B 0.000,C 180.000} C_DIS
LIN {X 93.500,Y 83.046,Z 63.500,A 180.000,B 0.000,C 180.000} C_DIS
LIN {X 93.321,Y 83.094,Z 63.500,A 180.000,B 0.000,C 180.000} C_DIS
LIN {X 93.203,Y 83.131,Z 63.500,A 180.000,B 0.000,C 180.000} C_DIS
LIN {X 92.642,Y 83.310,Z 63.500,A 180.000,B 0.000,C 180.000} C_DIS
LIN {X 92.606,Y 83.322,Z 63.500,A 180.000,B 0.000,C 180.000} C_DIS
LIN {X 92.427,Y 83.386,Z 63.500,A 180.000,B 0.000,C 180.000} C_DIS
LIN {X 91.891,Y 83.591,Z 63.500,A 180.000,B 0.000,C 180.000} C_DIS
LIN {X 91.712,Y 83.662,Z 63.500,A 180.000,B 0.000,C 180.000} C_DIS
LIN {X 91.700,Y 83.668,Z 63.500,A 180.000,B 0.000,C 180.000} C_DIS
LIN {X 91.176,Y 83.902,Z 63.500,A 180.000,B 0.000,C 180.000} C_DIS
LIN {X 90.997,Y 83.983,Z 63.500,A 180.000,B 0.000,C 180.000} C_DIS
LIN {X 90.913,Y 84.025,Z 63.500,A 180.000,B 0.000,C 180.000} C_DIS
LIN {X 90.461,Y 84.259,Z 63.500,A 180.000,B 0.000,C 180.000} C_DIS
LIN {X 90.282,Y 84.351,Z 63.500,A 180.000,B 0.000,C 180.000} C_DIS
LIN {X 90.225,Y 84.383,Z 63.500,A 180.000,B 0.000,C 180.000} C_DIS
LIN {X 90.103,Y 84.454,Z 63.500,A 180.000,B 0.000,C 180.000} C_DIS
LIN {X 89.618,Y 84.740,Z 63.500,A 180.000,B 0.000,C 180.000} C_DIS
LIN {X 89.567,Y 84.770,Z 63.500,A 180.000,B 0.000,C 180.000} C_DIS
LIN {X 89.388,Y 84.886,Z 63.500,A 180.000,B 0.000,C 180.000} C_DIS
LIN {X 89.031,Y 85.125,Z 63.500,A 180.000,B 0.000,C 180.000} C_DIS
LIN {X 88.852,Y 85.244,Z 63.500,A 180.000,B 0.000,C 180.000} C_DIS
LIN {X 88.806,Y 85.276,Z 63.500,A 180.000,B 0.000,C 180.000} C_DIS
LIN {X 88.673,Y 85.376,Z 63.500,A 180.000,B 0.000,C 180.000} C_DIS
LIN {X 88.316,Y 85.645,Z 63.500,A 180.000,B 0.000,C 180.000} C_DIS
LIN {X 88.137,Y 85.781,Z 63.500,A 180.000,B 0.000,C 180.000} C_DIS
LIN {X 88.098,Y 85.813,Z 63.500,A 180.000,B 0.000,C 180.000} C_DIS
LIN {X 87.779,Y 86.082,Z 63.500,A 180.000,B 0.000,C 180.000} C_DIS
LIN {X 87.601,Y 86.233,Z 63.500,A 180.000,B 0.000,C 180.000} C_DIS
LIN {X 87.468,Y 86.349,Z 63.500,A 180.000,B 0.000,C 180.000} C_DIS
LIN {X 87.422,Y 86.393,Z 63.500,A 180.000,B 0.000,C 180.000} C_DIS
LIN {X 87.064,Y 86.731,Z 63.500,A 180.000,B 0.000,C 180.000} C_DIS
LIN {X 86.901,Y 86.885,Z 63.500,A 180.000,B 0.000,C 180.000} C_DIS
LIN {X 86.885,Y 86.901,Z 63.500,A 180.000,B 0.000,C 180.000} C_DIS
LIN {X 86.731,Y 87.064,Z 63.500,A 180.000,B 0.000,C 180.000} C_DIS
LIN {X 86.393,Y 87.422,Z 63.500,A 180.000,B 0.000,C 180.000} C_DIS
LIN {X 86.349,Y 87.468,Z 63.500,A 180.000,B 0.000,C 180.000} C_DIS
LIN {X 86.233,Y 87.601,Z 63.500,A 180.000,B 0.000,C 180.000} C_DIS
LIN {X 85.931,Y 87.958,Z 63.500,A 180.000,B 0.000,C 180.000} C_DIS
LIN {X 85.813,Y 88.098,Z 63.500,A 180.000,B 0.000,C 180.000} C_DIS
LIN {X 85.781,Y 88.137,Z 63.500,A 180.000,B 0.000,C 180.000} C_DIS
LIN {X 85.645,Y 88.316,Z 63.500,A 180.000,B 0.000,C 180.000} C_DIS
LIN {X 85.376,Y 88.673,Z 63.500,A 180.000,B 0.000,C 180.000} C_DIS
LIN {X 85.276,Y 88.806,Z 63.500,A 180.000,B 0.000,C 180.000} C_DIS
LIN {X 85.244,Y 88.852,Z 63.500,A 180.000,B 0.000,C 180.000} C_DIS
LIN {X 85.125,Y 89.031,Z 63.500,A 180.000,B 0.000,C 180.000} C_DIS
LIN {X 84.886,Y 89.388,Z 63.500,A 180.000,B 0.000,C 180.000} C_DIS
LIN {X 84.770,Y 89.567,Z 63.500,A 180.000,B 0.000,C 180.000} C_DIS
LIN {X 84.740,Y 89.618,Z 63.500,A 180.000,B 0.000,C 180.000} C_DIS
LIN {X 84.454,Y 90.103,Z 63.500,A 180.000,B 0.000,C 180.000} C_DIS
LIN {X 84.383,Y 90.225,Z 63.500,A 180.000,B 0.000,C 180.000} C_DIS
LIN {X 84.351,Y 90.282,Z 63.500,A 180.000,B 0.000,C 180.000} C_DIS
LIN {X 84.259,Y 90.461,Z 63.500,A 180.000,B 0.000,C 180.000} C_DIS
LIN {X 84.025,Y 90.913,Z 63.500,A 180.000,B 0.000,C 180.000} C_DIS
LIN {X 83.983,Y 90.997,Z 63.500,A 180.000,B 0.000,C 180.000} C_DIS
LIN {X 83.902,Y 91.176,Z 63.500,A 180.000,B 0.000,C 180.000} C_DIS
LIN {X 83.668,Y 91.700,Z 63.500,A 180.000,B 0.000,C 180.000} C_DIS
LIN {X 83.662,Y 91.712,Z 63.500,A 180.000,B 0.000,C 180.000} C_DIS
LIN {X 83.591,Y 91.891,Z 63.500,A 180.000,B 0.000,C 180.000} C_DIS
LIN {X 83.386,Y 92.427,Z 63.500,A 180.000,B 0.000,C 180.000} C_DIS
LIN {X 83.322,Y 92.606,Z 63.500,A 180.000,B 0.000,C 180.000} C_DIS
LIN {X 83.310,Y 92.642,Z 63.500,A 180.000,B 0.000,C 180.000} C_DIS
LIN {X 83.131,Y 93.203,Z 63.500,A 180.000,B 0.000,C 180.000} C_DIS
LIN {X 83.094,Y 93.321,Z 63.500,A 180.000,B 0.000,C 180.000} C_DIS
LIN {X 83.046,Y 93.500,Z 63.500,A 180.000,B 0.000,C 180.000} C_DIS
LIN {X 82.908,Y 94.036,Z 63.500,A 180.000,B 0.000,C 180.000} C_DIS
LIN {X 82.865,Y 94.215,Z 63.500,A 180.000,B 0.000,C 180.000} C_DIS
LIN {X 82.833,Y 94.374,Z 63.500,A 180.000,B 0.000,C 180.000} C_DIS
LIN {X 82.829,Y 94.394,Z 63.500,A 180.000,B 0.000,C 180.000} C_DIS
LIN {X 82.758,Y 94.751,Z 63.500,A 180.000,B 0.000,C 180.000} C_DIS
LIN {X 82.722,Y 94.930,Z 63.500,A 180.000,B 0.000,C 180.000} C_DIS
LIN {X 82.694,Y 95.109,Z 63.500,A 180.000,B 0.000,C 180.000} C_DIS
LIN {X 82.618,Y 95.645,Z 63.500,A 180.000,B 0.000,C 180.000} C_DIS
LIN {X 82.595,Y 95.815,Z 63.500,A 180.000,B 0.000,C 180.000} C_DIS
LIN {X 82.594,Y 95.824,Z 63.500,A 180.000,B 0.000,C 180.000} C_DIS
LIN {X 82.578,Y 96.003,Z 63.500,A 180.000,B 0.000,C 180.000} C_DIS
LIN {X 82.533,Y 96.539,Z 63.500,A 180.000,B 0.000,C 180.000} C_DIS
LIN {X 82.521,Y 96.718,Z 63.500,A 180.000,B 0.000,C 180.000} C_DIS
LIN {X 82.516,Y 96.897,Z 63.500,A 180.000,B 0.000,C 180.000} C_DIS
LIN {X 82.501,Y 97.433,Z 63.500,A 180.000,B 0.000,C 180.000} C_DIS
LIN {X 82.502,Y 97.612,Z 63.500,A 180.000,B 0.000,C 180.000} C_DIS
LIN {X 82.517,Y 98.148,Z 63.500,A 180.000,B 0.000,C 180.000} C_DIS
LIN {X 82.523,Y 98.327,Z 63.500,A 180.000,B 0.000,C 180.000} C_DIS
LIN {X 82.536,Y 98.505,Z 63.500,A 180.000,B 0.000,C 180.000} C_DIS
LIN {X 82.582,Y 99.042,Z 63.500,A 180.000,B 0.000,C 180.000} C_DIS
LIN {X 82.595,Y 99.185,Z 63.500,A 180.000,B 0.000,C 180.000} C_DIS
LIN {X 82.599,Y 99.221,Z 63.500,A 180.000,B 0.000,C 180.000} C_DIS
LIN {X 82.624,Y 99.399,Z 63.500,A 180.000,B 0.000,C 180.000} C_DIS
LIN {X 82.700,Y 99.936,Z 63.500,A 180.000,B 0.000,C 180.000} C_DIS
LIN {X 82.731,Y 100.114,Z 63.500,A 180.000,B 0.000,C 180.000} C_DIS
LIN {X 82.838,Y 100.651,Z 63.500,A 180.000,B 0.000,C 180.000} C_DIS
LIN {X 82.874,Y 100.829,Z 63.500,A 180.000,B 0.000,C 180.000} C_DIS
LIN {X 82.919,Y 101.008,Z 63.500,A 180.000,B 0.000,C 180.000} C_DIS
LIN {X 83.057,Y 101.545,Z 63.500,A 180.000,B 0.000,C 180.000} C_DIS
LIN {X 83.108,Y 101.723,Z 63.500,A 180.000,B 0.000,C 180.000} C_DIS
LIN {X 83.310,Y 102.358,Z 63.500,A 180.000,B 0.000,C 180.000} C_DIS
LIN {X 83.336,Y 102.438,Z 63.500,A 180.000,B 0.000,C 180.000} C_DIS
LIN {X 83.403,Y 102.617,Z 63.500,A 180.000,B 0.000,C 180.000} C_DIS
LIN {X 83.608,Y 103.153,Z 63.500,A 180.000,B 0.000,C 180.000} C_DIS
LIN {X 83.668,Y 103.300,Z 63.500,A 180.000,B 0.000,C 180.000} C_DIS
LIN {X 83.922,Y 103.869,Z 63.500,A 180.000,B 0.000,C 180.000} C_DIS
LIN {X 84.005,Y 104.047,Z 63.500,A 180.000,B 0.000,C 180.000} C_DIS
LIN {X 84.025,Y 104.087,Z 63.500,A 180.000,B 0.000,C 180.000} C_DIS
LIN {X 84.282,Y 104.584,Z 63.500,A 180.000,B 0.000,C 180.000} C_DIS
LIN {X 84.375,Y 104.762,Z 63.500,A 180.000,B 0.000,C 180.000} C_DIS
LIN {X 84.383,Y 104.775,Z 63.500,A 180.000,B 0.000,C 180.000} C_DIS
LIN {X 84.480,Y 104.941,Z 63.500,A 180.000,B 0.000,C 180.000} C_DIS
LIN {X 84.740,Y 105.382,Z 63.500,A 180.000,B 0.000,C 180.000} C_DIS
LIN {X 84.797,Y 105.477,Z 63.500,A 180.000,B 0.000,C 180.000} C_DIS
LIN {X 84.915,Y 105.656,Z 63.500,A 180.000,B 0.000,C 180.000} C_DIS
LIN {X 85.154,Y 106.014,Z 63.500,A 180.000,B 0.000,C 180.000} C_DIS
LIN {X 85.276,Y 106.193,Z 63.500,A 180.000,B 0.000,C 180.000} C_DIS
LIN {X 85.276,Y 106.194,Z 63.500,A 180.000,B 0.000,C 180.000} C_DIS
LIN {X 85.409,Y 106.371,Z 63.500,A 180.000,B 0.000,C 180.000} C_DIS
LIN {X 85.678,Y 106.729,Z 63.500,A 180.000,B 0.000,C 180.000} C_DIS
LIN {X 85.813,Y 106.902,Z 63.500,A 180.000,B 0.000,C 180.000} C_DIS
LIN {X 85.818,Y 106.908,Z 63.500,A 180.000,B 0.000,C 180.000} C_DIS
LIN {X 86.271,Y 107.444,Z 63.500,A 180.000,B 0.000,C 180.000} C_DIS
LIN {X 86.349,Y 107.532,Z 63.500,A 180.000,B 0.000,C 180.000} C_DIS
LIN {X 86.435,Y 107.623,Z 63.500,A 180.000,B 0.000,C 180.000} C_DIS
LIN {X 86.773,Y 107.980,Z 63.500,A 180.000,B 0.000,C 180.000} C_DIS
LIN {X 86.885,Y 108.099,Z 63.500,A 180.000,B 0.000,C 180.000} C_DIS
LIN {X 86.947,Y 108.159,Z 63.500,A 180.000,B 0.000,C 180.000} C_DIS
LIN {X 87.422,Y 108.607,Z 63.500,A 180.000,B 0.000,C 180.000} C_DIS
LIN {X 87.517,Y 108.695,Z 63.500,A 180.000,B 0.000,C 180.000} C_DIS
LIN {X 87.601,Y 108.767,Z 63.500,A 180.000,B 0.000,C 180.000} C_DIS
LIN {X 87.958,Y 109.069,Z 63.500,A 180.000,B 0.000,C 180.000} C_DIS
LIN {X 88.137,Y 109.219,Z 63.500,A 180.000,B 0.000,C 180.000} C_DIS
LIN {X 88.153,Y 109.232,Z 63.500,A 180.000,B 0.000,C 180.000} C_DIS
LIN {X 88.316,Y 109.355,Z 63.500,A 180.000,B 0.000,C 180.000} C_DIS
LIN {X 88.673,Y 109.624,Z 63.500,A 180.000,B 0.000,C 180.000} C_DIS
LIN {X 88.852,Y 109.756,Z 63.500,A 180.000,B 0.000,C 180.000} C_DIS
LIN {X 88.870,Y 109.768,Z 63.500,A 180.000,B 0.000,C 180.000} C_DIS
LIN {X 89.031,Y 109.875,Z 63.500,A 180.000,B 0.000,C 180.000} C_DIS
LIN {X 89.405,Y 110.126,Z 63.500,A 180.000,B 0.000,C 180.000} C_DIS
LIN {X 89.567,Y 110.230,Z 63.500,A 180.000,B 0.000,C 180.000} C_DIS
LIN {X 89.693,Y 110.304,Z 63.500,A 180.000,B 0.000,C 180.000} C_DIS
LIN {X 90.103,Y 110.546,Z 63.500,A 180.000,B 0.000,C 180.000} C_DIS
LIN {X 90.282,Y 110.649,Z 63.500,A 180.000,B 0.000,C 180.000} C_DIS
LIN {X 90.307,Y 110.662,Z 63.500,A 180.000,B 0.000,C 180.000} C_DIS
LIN {X 90.818,Y 110.926,Z 63.500,A 180.000,B 0.000,C 180.000} C_DIS
LIN {X 90.997,Y 111.017,Z 63.500,A 180.000,B 0.000,C 180.000} C_DIS
LIN {X 91.002,Y 111.019,Z 63.500,A 180.000,B 0.000,C 180.000} C_DIS
LIN {X 91.176,Y 111.098,Z 63.500,A 180.000,B 0.000,C 180.000} C_DIS
LIN {X 91.533,Y 111.258,Z 63.500,A 180.000,B 0.000,C 180.000} C_DIS
LIN {X 91.712,Y 111.338,Z 63.500,A 180.000,B 0.000,C 180.000} C_DIS
LIN {X 91.806,Y 111.377,Z 63.500,A 180.000,B 0.000,C 180.000} C_DIS
LIN {X 91.891,Y 111.409,Z 63.500,A 180.000,B 0.000,C 180.000} C_DIS
LIN {X 92.427,Y 111.614,Z 63.500,A 180.000,B 0.000,C 180.000} C_DIS
LIN {X 92.606,Y 111.678,Z 63.500,A 180.000,B 0.000,C 180.000} C_DIS
LIN {X 92.964,Y 111.792,Z 63.500,A 180.000,B 0.000,C 180.000} C_DIS
LIN {X 93.142,Y 111.849,Z 63.500,A 180.000,B 0.000,C 180.000} C_DIS
LIN {X 93.321,Y 111.906,Z 63.500,A 180.000,B 0.000,C 180.000} C_DIS
LIN {X 93.346,Y 111.913,Z 63.500,A 180.000,B 0.000,C 180.000} C_DIS
LIN {X 93.500,Y 111.954,Z 63.500,A 180.000,B 0.000,C 180.000} C_DIS
LIN {X 94.036,Y 112.092,Z 63.500,A 180.000,B 0.000,C 180.000} C_DIS
LIN {X 94.215,Y 112.135,Z 63.500,A 180.000,B 0.000,C 180.000} C_DIS
LIN {X 94.394,Y 112.171,Z 63.500,A 180.000,B 0.000,C 180.000} C_DIS
LIN {X 94.895,Y 112.271,Z 63.500,A 180.000,B 0.000,C 180.000} C_DIS
LIN {X 94.930,Y 112.278,Z 63.500,A 180.000,B 0.000,C 180.000} C_DIS
LIN {X 95.109,Y 112.306,Z 63.500,A 180.000,B 0.000,C 180.000} C_DIS
LIN {X 95.645,Y 112.382,Z 63.500,A 180.000,B 0.000,C 180.000} C_DIS
LIN {X 95.824,Y 112.406,Z 63.500,A 180.000,B 0.000,C 180.000} C_DIS
LIN {X 96.003,Y 112.422,Z 63.500,A 180.000,B 0.000,C 180.000} C_DIS
LIN {X 96.539,Y 112.467,Z 63.500,A 180.000,B 0.000,C 180.000} C_DIS
LIN {X 96.718,Y 112.479,Z 63.500,A 180.000,B 0.000,C 180.000} C_DIS
LIN {X 96.897,Y 112.484,Z 63.500,A 180.000,B 0.000,C 180.000} C_DIS
LIN {X 97.433,Y 112.499,Z 63.500,A 180.000,B 0.000,C 180.000} C_DIS
LIN {X 97.612,Y 112.498,Z 63.500,A 180.000,B 0.000,C 180.000} C_DIS
LIN {X 98.148,Y 112.483,Z 63.500,A 180.000,B 0.000,C 180.000} C_DIS
LIN {X 98.327,Y 112.477,Z 63.500,A 180.000,B 0.000,C 180.000} C_DIS
LIN {X 98.505,Y 112.464,Z 63.500,A 180.000,B 0.000,C 180.000} C_DIS
LIN {X 99.042,Y 112.418,Z 63.500,A 180.000,B 0.000,C 180.000} C_DIS
LIN {X 99.221,Y 112.401,Z 63.500,A 180.000,B 0.000,C 180.000} C_DIS
LIN {X 99.399,Y 112.376,Z 63.500,A 180.000,B 0.000,C 180.000} C_DIS
LIN {X 99.936,Y 112.300,Z 63.500,A 180.000,B 0.000,C 180.000} C_DIS
LIN {X 100.105,Y 112.271,Z 63.500,A 180.000,B 0.000,C 180.000} C_DIS
LIN {X 100.651,Y 112.162,Z 63.500,A 180.000,B 0.000,C 180.000} C_DIS
LIN {X 100.829,Y 112.126,Z 63.500,A 180.000,B 0.000,C 180.000} C_DIS
LIN {X 100.966,Y 112.092,Z 63.500,A 180.000,B 0.000,C 180.000} C_DIS
LIN {X 101.545,Y 111.943,Z 63.500,A 180.000,B 0.000,C 180.000} C_DIS
LIN {X 101.654,Y 111.913,Z 63.500,A 180.000,B 0.000,C 180.000} C_DIS
LIN {X 101.723,Y 111.892,Z 63.500,A 180.000,B 0.000,C 180.000} C_DIS
LIN {X 102.260,Y 111.721,Z 63.500,A 180.000,B 0.000,C 180.000} C_DIS
LIN {X 102.438,Y 111.664,Z 63.500,A 180.000,B 0.000,C 180.000} C_DIS
LIN {X 102.617,Y 111.597,Z 63.500,A 180.000,B 0.000,C 180.000} C_DIS
LIN {X 103.153,Y 111.392,Z 63.500,A 180.000,B 0.000,C 180.000} C_DIS
LIN {X 103.194,Y 111.377,Z 63.500,A 180.000,B 0.000,C 180.000} C_DIS
LIN {X 103.332,Y 111.318,Z 63.500,A 180.000,B 0.000,C 180.000} C_DIS
LIN {X 103.869,Y 111.078,Z 63.500,A 180.000,B 0.000,C 180.000} C_DIS
LIN {X 103.998,Y 111.019,Z 63.500,A 180.000,B 0.000,C 180.000} C_DIS
LIN {X 104.047,Y 110.995,Z 63.500,A 180.000,B 0.000,C 180.000} C_DIS
LIN {X 104.226,Y 110.903,Z 63.500,A 180.000,B 0.000,C 180.000} C_DIS
LIN {X 104.693,Y 110.662,Z 63.500,A 180.000,B 0.000,C 180.000} C_DIS
LIN {X 104.762,Y 110.625,Z 63.500,A 180.000,B 0.000,C 180.000} C_DIS
LIN {X 104.941,Y 110.520,Z 63.500,A 180.000,B 0.000,C 180.000} C_DIS
LIN {X 105.307,Y 110.304,Z 63.500,A 180.000,B 0.000,C 180.000} C_DIS
LIN {X 105.477,Y 110.203,Z 63.500,A 180.000,B 0.000,C 180.000} C_DIS
LIN {X 105.595,Y 110.126,Z 63.500,A 180.000,B 0.000,C 180.000} C_DIS
LIN {X 106.014,Y 109.846,Z 63.500,A 180.000,B 0.000,C 180.000} C_DIS
LIN {X 106.130,Y 109.768,Z 63.500,A 180.000,B 0.000,C 180.000} C_DIS
LIN {X 106.193,Y 109.724,Z 63.500,A 180.000,B 0.000,C 180.000} C_DIS
LIN {X 106.371,Y 109.591,Z 63.500,A 180.000,B 0.000,C 180.000} C_DIS
LIN {X 106.729,Y 109.322,Z 63.500,A 180.000,B 0.000,C 180.000} C_DIS
LIN {X 106.847,Y 109.232,Z 63.500,A 180.000,B 0.000,C 180.000} C_DIS
LIN {X 106.908,Y 109.182,Z 63.500,A 180.000,B 0.000,C 180.000} C_DIS
LIN {X 107.068,Y 109.046,Z 63.500,A 180.000,B 0.000,C 180.000} C_DIS
; Link Move Starts
LIN {X 107.309,Y 108.843,Z 63.500,A 180.000,B 0.000,C 180.000} C_DIS
LIN {X 107.547,Y 108.637,Z 63.499,A 180.000,B 0.000,C 180.000} C_DIS
LIN {X 107.776,Y 108.421,Z 63.498,A 180.000,B 0.000,C 180.000} C_DIS
LIN {X 108.005,Y 108.204,Z 63.496,A 180.000,B 0.000,C 180.000} C_DIS
LIN {X 108.227,Y 107.981,Z 63.494,A 180.000,B 0.000,C 180.000} C_DIS
LIN {X 108.443,Y 107.752,Z 63.491,A 180.000,B 0.000,C 180.000} C_DIS
LIN {X 108.659,Y 107.523,Z 63.488,A 180.000,B 0.000,C 180.000} C_DIS
LIN {X 108.864,Y 107.284,Z 63.485,A 180.000,B 0.000,C 180.000} C_DIS
LIN {X 109.068,Y 107.043,Z 63.481,A 180.000,B 0.000,C 180.000} C_DIS
LIN {X 109.268,Y 106.800,Z 63.477,A 180.000,B 0.000,C 180.000} C_DIS
LIN {X 109.457,Y 106.548,Z 63.472,A 180.000,B 0.000,C 180.000} C_DIS
LIN {X 109.552,Y 106.423,Z 63.469,A 180.000,B 0.000,C 180.000} C_DIS
LIN {X 109.647,Y 106.297,Z 63.467,A 180.000,B 0.000,C 180.000} C_DIS
LIN {X 109.740,Y 106.170,Z 63.464,A 180.000,B 0.000,C 180.000} C_DIS
LIN {X 109.829,Y 106.039,Z 63.461,A 180.000,B 0.000,C 180.000} C_DIS
LIN {X 109.916,Y 105.909,Z 63.459,A 180.000,B 0.000,C 180.000} C_DIS
LIN {X 110.004,Y 105.778,Z 63.456,A 180.000,B 0.000,C 180.000} C_DIS
LIN {X 110.091,Y 105.647,Z 63.452,A 180.000,B 0.000,C 180.000} C_DIS
LIN {X 110.178,Y 105.516,Z 63.449,A 180.000,B 0.000,C 180.000} C_DIS
LIN {X 110.261,Y 105.381,Z 63.446,A 180.000,B 0.000,C 180.000} C_DIS
LIN {X 110.341,Y 105.246,Z 63.443,A 180.000,B 0.000,C 180.000} C_DIS
LIN {X 110.421,Y 105.110,Z 63.439,A 180.000,B 0.000,C 180.000} C_DIS
LIN {X 110.501,Y 104.974,Z 63.436,A 180.000,B 0.000,C 180.000} C_DIS
LIN {X 110.581,Y 104.839,Z 63.432,A 180.000,B 0.000,C 180.000} C_DIS
LIN {X 110.658,Y 104.701,Z 63.428,A 180.000,B 0.000,C 180.000} C_DIS
LIN {X 110.730,Y 104.561,Z 63.425,A 180.000,B 0.000,C 180.000} C_DIS
LIN {X 110.802,Y 104.421,Z 63.421,A 180.000,B 0.000,C 180.000} C_DIS
LIN {X 110.875,Y 104.281,Z 63.417,A 180.000,B 0.000,C 180.000} C_DIS
LIN {X 110.947,Y 104.141,Z 63.413,A 180.000,B 0.000,C 180.000} C_DIS
LIN {X 111.018,Y 104.001,Z 63.409,A 180.000,B 0.000,C 180.000} C_DIS
LIN {X 111.083,Y 103.858,Z 63.405,A 180.000,B 0.000,C 180.000} C_DIS
LIN {X 111.147,Y 103.714,Z 63.400,A 180.000,B 0.000,C 180.000} C_DIS
LIN {X 111.212,Y 103.570,Z 63.396,A 180.000,B 0.000,C 180.000} C_DIS
LIN {X 111.276,Y 103.426,Z 63.392,A 180.000,B 0.000,C 180.000} C_DIS
LIN {X 111.340,Y 103.282,Z 63.387,A 180.000,B 0.000,C 180.000} C_DIS
LIN {X 111.399,Y 103.136,Z 63.383,A 180.000,B 0.000,C 180.000} C_DIS
LIN {X 111.455,Y 102.989,Z 63.378,A 180.000,B 0.000,C 180.000} C_DIS
LIN {X 111.511,Y 102.842,Z 63.373,A 180.000,B 0.000,C 180.000} C_DIS
LIN {X 111.567,Y 102.695,Z 63.369,A 180.000,B 0.000,C 180.000} C_DIS
LIN {X 111.624,Y 102.548,Z 63.364,A 180.000,B 0.000,C 180.000} C_DIS
LIN {X 111.677,Y 102.399,Z 63.359,A 180.000,B 0.000,C 180.000} C_DIS
LIN {X 111.725,Y 102.249,Z 63.354,A 180.000,B 0.000,C 180.000} C_DIS
LIN {X 111.748,Y 102.174,Z 63.351,A 180.000,B 0.000,C 180.000} C_DIS
LIN {X 111.772,Y 102.099,Z 63.349,A 180.000,B 0.000,C 180.000} C_DIS
LIN {X 111.796,Y 102.024,Z 63.346,A 180.000,B 0.000,C 180.000} C_DIS
LIN {X 111.820,Y 101.949,Z 63.344,A 180.000,B 0.000,C 180.000} C_DIS
LIN {X 111.844,Y 101.874,Z 63.341,A 180.000,B 0.000,C 180.000} C_DIS
LIN {X 111.868,Y 101.799,Z 63.339,A 180.000,B 0.000,C 180.000} C_DIS
LIN {X 111.892,Y 101.724,Z 63.336,A 180.000,B 0.000,C 180.000} C_DIS
LIN {X 111.915,Y 101.649,Z 63.333,A 180.000,B 0.000,C 180.000} C_DIS
LIN {X 111.935,Y 101.573,Z 63.331,A 180.000,B 0.000,C 180.000} C_DIS
LIN {X 111.975,Y 101.420,Z 63.325,A 180.000,B 0.000,C 180.000} C_DIS
LIN {X 112.014,Y 101.268,Z 63.320,A 180.000,B 0.000,C 180.000} C_DIS
LIN {X 112.053,Y 101.115,Z 63.315,A 180.000,B 0.000,C 180.000} C_DIS
LIN {X 112.093,Y 100.963,Z 63.309,A 180.000,B 0.000,C 180.000} C_DIS
LIN {X 112.112,Y 100.886,Z 63.306,A 180.000,B 0.000,C 180.000} C_DIS
LIN {X 112.130,Y 100.810,Z 63.304,A 180.000,B 0.000,C 180.000} C_DIS
LIN {X 112.146,Y 100.733,Z 63.301,A 180.000,B 0.000,C 180.000} C_DIS
LIN {X 112.192,Y 100.501,Z 63.293,A 180.000,B 0.000,C 180.000} C_DIS
LIN {X 112.223,Y 100.346,Z 63.287,A 180.000,B 0.000,C 180.000} C_DIS
LIN {X 112.238,Y 100.269,Z 63.285,A 180.000,B 0.000,C 180.000} C_DIS
LIN {X 112.269,Y 100.115,Z 63.279,A 180.000,B 0.000,C 180.000} C_DIS
LIN {X 112.284,Y 100.037,Z 63.276,A 180.000,B 0.000,C 180.000} C_DIS
LIN {X 112.296,Y 99.960,Z 63.274,A 180.000,B 0.000,C 180.000} C_DIS
LIN {X 112.308,Y 99.882,Z 63.271,A 180.000,B 0.000,C 180.000} C_DIS
LIN {X 112.330,Y 99.726,Z 63.265,A 180.000,B 0.000,C 180.000} C_DIS
LIN {X 112.341,Y 99.648,Z 63.263,A 180.000,B 0.000,C 180.000} C_DIS
